LIN {X 0,Y 253.688,Z 332.355,A -85,B 0,C 180,E1 -18838.131,E2 -18838.131} C_VEL
LIN {X 0,Y 253.519,Z 331.287,A -85,B 0,C 180,E1 -18838.229,E2 -18838.229} C_VEL
LIN {X 0,Y 251.232,Z 319.885,A -85,B 0,C 180,E1 -18842.107,E2 -18842.107} C_VEL
LIN {X 0,Y 249.083,Z 309.456,A -85,B 0,C 180,E1 -18845.847,E2 -18845.847} C_VEL
LIN {X 0,Y 248.969,Z 309.472,A -85,B 0,C 180,E1 -18850.484,E2 -18850.484} C_VEL
LIN {X 0,Y 248.957,Z 309.474,A -85,B 0,C 180,E1 -18854.887,E2 -18854.887} C_VEL
LIN {X 0,Y 248.971,Z 309.47,A -85,B 0,C 180,E1 -18857.352,E2 -18857.352} C_VEL
LIN {X 0,Y 249.037,Z 309.461,A -85,B 0,C 180,E1 -18862.199,E2 -18862.199} C_VEL
LIN {X 0,Y 249.034,Z 309.462,A -85,B 0,C 180,E1 -18865.637,E2 -18865.637} C_VEL
LIN {X 0,Y 248.989,Z 309.469,A -85,B 0,C 180,E1 -18869.464,E2 -18869.464} C_VEL
LIN {X 0,Y 249.025,Z 309.467,A -85,B 0,C 180,E1 -18873.156,E2 -18873.156} C_VEL
LIN {X 0,Y 249.039,Z 309.461,A -85,B 0,C 180,E1 -18876.728,E2 -18876.728} C_VEL
LIN {X 0,Y 249.043,Z 309.46,A -85,B 0,C 180,E1 -18880.205,E2 -18880.205} C_VEL
LIN {X 0,Y 249.146,Z 309.448,A -85,B 0,C 180,E1 -18883.615,E2 -18883.615} C_VEL
LIN {X 0,Y 249.209,Z 309.44,A -85,B 0,C 180,E1 -18888.614,E2 -18888.614} C_VEL
LIN {X 0,Y 249.431,Z 309.412,A -85,B 0,C 180,E1 -18891.9,E2 -18891.9} C_VEL
LIN {X 0,Y 249.266,Z 309.434,A -85,B 0,C 180,E1 -18895.147,E2 -18895.147} C_VEL
LIN {X 0,Y 249.653,Z 309.385,A -85,B 0,C 180,E1 -18898.386,E2 -18898.386} C_VEL
LIN {X 0,Y 249.653,Z 309.386,A -85,B 0,C 180,E1 -18901.612,E2 -18901.612} C_VEL
LIN {X 0,Y 249.41,Z 309.413,A -85,B 0,C 180,E1 -18906.803,E2 -18906.803} C_VEL
LIN {X 0,Y 249.32,Z 309.427,A -85,B 0,C 180,E1 -18909.737,E2 -18909.737} C_VEL
LIN {X 0,Y 249.153,Z 309.447,A -85,B 0,C 180,E1 -18914.706,E2 -18914.706} C_VEL
LIN {X 0,Y 249.067,Z 309.457,A -85,B 0,C 180,E1 -18918.082,E2 -18918.082} C_VEL
LIN {X 0,Y 249.032,Z 309.464,A -85,B 0,C 180,E1 -18921.522,E2 -18921.522} C_VEL
LIN {X 0,Y 249.103,Z 309.455,A -85,B 0,C 180,E1 -18925.475,E2 -18925.475} C_VEL
LIN {X 0,Y 249.061,Z 309.457,A -85,B 0,C 180,E1 -18928.989,E2 -18928.989} C_VEL
LIN {X 0,Y 249.019,Z 309.464,A -85,B 0,C 180,E1 -18932.426,E2 -18932.426} C_VEL
LIN {X 0,Y 249.043,Z 309.461,A -85,B 0,C 180,E1 -18936.342,E2 -18936.342} C_VEL
LIN {X 0,Y 248.997,Z 309.467,A -85,B 0,C 180,E1 -18940.479,E2 -18940.479} C_VEL
LIN {X 0,Y 249.004,Z 309.464,A -85,B 0,C 180,E1 -18944.878,E2 -18944.878} C_VEL
LIN {X 0,Y 249.05,Z 309.46,A -85,B 0,C 180,E1 -18947.372,E2 -18947.372} C_VEL
LIN {X 0,Y 249.046,Z 309.46,A -85,B 0,C 180,E1 -18951.624,E2 -18951.624} C_VEL
LIN {X 0,Y 249.057,Z 309.459,A -85,B 0,C 180,E1 -18955.642,E2 -18955.642} C_VEL
LIN {X 0,Y 249.043,Z 309.46,A -85,B 0,C 180,E1 -18959.472,E2 -18959.472} C_VEL
LIN {X 0,Y 249.068,Z 309.457,A -85,B 0,C 180,E1 -18963.162,E2 -18963.162} C_VEL
LIN {X 0,Y 249.078,Z 309.457,A -85,B 0,C 180,E1 -18966.732,E2 -18966.732} C_VEL
LIN {X 0,Y 249.11,Z 309.453,A -85,B 0,C 180,E1 -18970.211,E2 -18970.211} C_VEL
LIN {X 0,Y 249.24,Z 309.436,A -85,B 0,C 180,E1 -18973.621,E2 -18973.621} C_VEL
LIN {X 0,Y 249.251,Z 309.437,A -85,B 0,C 180,E1 -18978.615,E2 -18978.615} C_VEL
LIN {X 0,Y 249.483,Z 309.406,A -85,B 0,C 180,E1 -18981.901,E2 -18981.901} C_VEL
LIN {X 0,Y 249.434,Z 309.414,A -85,B 0,C 180,E1 -18986.767,E2 -18986.767} C_VEL
LIN {X 0,Y 249.726,Z 309.376,A -85,B 0,C 180,E1 -18989.997,E2 -18989.997} C_VEL
LIN {X 0,Y 249.434,Z 309.411,A -85,B 0,C 180,E1 -18993.228,E2 -18993.228} C_VEL
LIN {X 0,Y 249.479,Z 309.407,A -85,B 0,C 180,E1 -18998.094,E2 -18998.094} C_VEL
LIN {X 0,Y 249.248,Z 309.435,A -85,B 0,C 180,E1 -19001.38,E2 -19001.38} C_VEL
LIN {X 0,Y 249.234,Z 309.437,A -85,B 0,C 180,E1 -19006.374,E2 -19006.374} C_VEL
LIN {X 0,Y 249.125,Z 309.451,A -85,B 0,C 180,E1 -19011.51,E2 -19011.51} C_VEL
LIN {X 0,Y 249.119,Z 309.452,A -85,B 0,C 180,E1 -19015.478,E2 -19015.478} C_VEL
LIN {X 0,Y 249.069,Z 309.461,A -85,B 0,C 180,E1 -19018.989,E2 -19018.989} C_VEL
LIN {X 0,Y 249.08,Z 309.458,A -85,B 0,C 180,E1 -19023.799,E2 -19023.799} C_VEL
LIN {X 0,Y 252.845,Z 319.658,A -85,B 0,C 180,E1 -19024.515,E2 -19024.515} C_VEL
LIN {X 0,Y 259.68,Z 338.346,A -85,B 0,C 180,E1 -19025.737,E2 -19025.737} C_VEL
LIN {X 0,Y 260.257,Z 340.087,A -85,B 0,C 180,E1 -19025.842,E2 -19025.842} C_VEL
LIN {X 0,Y 257.273,Z 412.228,A -85,B 0,C 180,E1 -19028.37,E2 -19028.37} C_VEL
LIN {X 0,Y 256.65,Z 424.844,A -85,B 0,C 180,E1 -19029.098,E2 -19029.098} C_VEL
LIN {X 0,Y 255.648,Z 437.472,A -85,B 0,C 180,E1 -19030.113,E2 -19030.113} C_VEL
LIN {X 0,Y 254.445,Z 449.649,A -85,B 0,C 180,E1 -19031.423,E2 -19031.423} C_VEL
LIN {X 0,Y 253.15,Z 460.66,A -85,B 0,C 180,E1 -19032.928,E2 -19032.928} C_VEL
LIN {X 0,Y 251.959,Z 470.882,A -85,B 0,C 180,E1 -19034.662,E2 -19034.662} C_VEL
LIN {X 0,Y 250.599,Z 481.033,A -85,B 0,C 180,E1 -19036.807,E2 -19036.807} C_VEL
LIN {X 0,Y 249.471,Z 489.721,A -85,B 0,C 180,E1 -19039.082,E2 -19039.082} C_VEL
LIN {X 0,Y 248.537,Z 497.225,A -85,B 0,C 180,E1 -19041.531,E2 -19041.531} C_VEL
LIN {X 0,Y 247.852,Z 503.12,A -85,B 0,C 180,E1 -19043.96,E2 -19043.96} C_VEL
LIN {X 0,Y 247.453,Z 507.724,A -85,B 0,C 180,E1 -19046.371,E2 -19046.371} C_VEL
LIN {X 0,Y 247.04,Z 511.734,A -85,B 0,C 180,E1 -19049.199,E2 -19049.199} C_VEL
LIN {X 0,Y 246.904,Z 514.316,A -85,B 0,C 180,E1 -19051.917,E2 -19051.917} C_VEL
LIN {X 0,Y 247.262,Z 515.891,A -85,B 0,C 180,E1 -19055.423,E2 -19055.423} C_VEL
LIN {X 0,Y 247.98,Z 515.755,A -85,B 0,C 180,E1 -19058.382,E2 -19058.382} C_VEL
LIN {X 0,Y 248.621,Z 515,A -85,B 0,C 180,E1 -19060.172,E2 -19060.172} C_VEL
LIN {X 0,Y 249.915,Z 512.823,A -85,B 0,C 180,E1 -19062.939,E2 -19062.939} C_VEL
LIN {X 0,Y 251.501,Z 509.738,A -85,B 0,C 180,E1 -19065.435,E2 -19065.435} C_VEL
LIN {X 0,Y 253.476,Z 505.327,A -85,B 0,C 180,E1 -19067.999,E2 -19067.999} C_VEL
LIN {X 0,Y 255.951,Z 499.537,A -85,B 0,C 180,E1 -19070.518,E2 -19070.518} C_VEL
LIN {X 0,Y 258.79,Z 492.2,A -85,B 0,C 180,E1 -19072.981,E2 -19072.981} C_VEL
LIN {X 0,Y 261.491,Z 484.692,A -85,B 0,C 180,E1 -19074.979,E2 -19074.979} C_VEL
LIN {X 0,Y 264.556,Z 475.406,A -85,B 0,C 180,E1 -19076.955,E2 -19076.955} C_VEL
LIN {X 0,Y 267.336,Z 465.509,A -85,B 0,C 180,E1 -19078.655,E2 -19078.655} C_VEL
LIN {X 0,Y 270.129,Z 454.102,A -85,B 0,C 180,E1 -19080.187,E2 -19080.187} C_VEL
LIN {X 0,Y 272.685,Z 441.841,A -85,B 0,C 180,E1 -19081.478,E2 -19081.478} C_VEL
LIN {X 0,Y 274.666,Z 429.131,A -85,B 0,C 180,E1 -19082.484,E2 -19082.484} C_VEL
LIN {X 0,Y 276.268,Z 415.345,A -85,B 0,C 180,E1 -19083.248,E2 -19083.248} C_VEL
LIN {X 0,Y 281,Z 357.266,A -85,B 0,C 180,E1 -19085.293,E2 -19085.293} C_VEL
LIN {X 0,Y 277.332,Z 349.628,A -85,B 0,C 180,E1 -19086.613,E2 -19086.613} C_VEL
LIN {X 0,Y 276.385,Z 347.949,A -85,B 0,C 180,E1 -19086.951,E2 -19086.951} C_VEL
LIN {X 0,Y 274.604,Z 345.866,A -85,B 0,C 180,E1 -19087.543,E2 -19087.543} C_VEL
LIN {X 0,Y 270.87,Z 344.364,A -85,B 0,C 180,E1 -19088.684,E2 -19088.684} C_VEL
LIN {X 0,Y 267.23,Z 343.003,A -85,B 0,C 180,E1 -19089.882,E2 -19089.882} C_VEL
LIN {X 0,Y 265.578,Z 341.11,A -85,B 0,C 180,E1 -19090.553,E2 -19090.553} C_VEL
LIN {X 0,Y 262.045,Z 336.05,A -85,B 0,C 180,E1 -19092.207,E2 -19092.207} C_VEL
LIN {X 0,Y 258.278,Z 331.025,A -85,B 0,C 180,E1 -19094.177,E2 -19094.177} C_VEL
LIN {X 0,Y 254.479,Z 326.181,A -85,B 0,C 180,E1 -19096.472,E2 -19096.472} C_VEL
LIN {X 0,Y 251.933,Z 323.447,A -85,B 0,C 180,E1 -19098.228,E2 -19098.228} C_VEL
LIN {X 0,Y 248.642,Z 319.476,A -85,B 0,C 180,E1 -19101.152,E2 -19101.152} C_VEL
LIN {X 0,Y 244.923,Z 316.459,A -85,B 0,C 180,E1 -19106.218,E2 -19106.218} C_VEL
LIN {X 0,Y 244.041,Z 315.707,A -85,B 0,C 180,E1 -19109.432,E2 -19109.432} C_VEL
LIN {X 0,Y 244.605,Z 316.843,A -85,B 0,C 180,E1 -19113.582,E2 -19113.582} C_VEL
LIN {X 0,Y 245.437,Z 318.272,A -85,B 0,C 180,E1 -19116.185,E2 -19116.185} C_VEL
LIN {X 0,Y 248.579,Z 323.493,A -85,B 0,C 180,E1 -19120.431,E2 -19120.431} C_VEL
LIN {X 0,Y 251.56,Z 327.54,A -85,B 0,C 180,E1 -19123.051,E2 -19123.051} C_VEL
LIN {X 0,Y 256.502,Z 335.172,A -85,B 0,C 180,E1 -19126.428,E2 -19126.428} C_VEL
LIN {X 0,Y 260.53,Z 342.026,A -85,B 0,C 180,E1 -19128.71,E2 -19128.71} C_VEL
LIN {X 0,Y 263.954,Z 348.304,A -85,B 0,C 180,E1 -19130.433,E2 -19130.433} C_VEL
LIN {X 0,Y 267.188,Z 354.826,A -85,B 0,C 180,E1 -19131.92,E2 -19131.92} C_VEL
LIN {X 0,Y 270.159,Z 361.496,A -85,B 0,C 180,E1 -19133.236,E2 -19133.236} C_VEL
LIN {X 0,Y 272.398,Z 367.573,A -85,B 0,C 180,E1 -19134.204,E2 -19134.204} C_VEL
LIN {X 0,Y 273.727,Z 381.745,A -85,B 0,C 180,E1 -19135.364,E2 -19135.364} C_VEL
LIN {X 0,Y 274.04,Z 390.294,A -85,B 0,C 180,E1 -19135.927,E2 -19135.927} C_VEL
LIN {X 0,Y 269.906,Z 437.588,A -85,B 0,C 180,E1 -19137.634,E2 -19137.634} C_VEL
LIN {X 0,Y 267.932,Z 451.025,A -85,B 0,C 180,E1 -19138.364,E2 -19138.364} C_VEL
LIN {X 0,Y 265.251,Z 463.95,A -85,B 0,C 180,E1 -19139.34,E2 -19139.34} C_VEL
LIN {X 0,Y 262.356,Z 475.61,A -85,B 0,C 180,E1 -19140.519,E2 -19140.519} C_VEL
LIN {X 0,Y 259.28,Z 486.361,A -85,B 0,C 180,E1 -19141.909,E2 -19141.909} C_VEL
LIN {X 0,Y 255.526,Z 498.244,A -85,B 0,C 180,E1 -19143.898,E2 -19143.898} C_VEL
LIN {X 0,Y 252.405,Z 507.111,A -85,B 0,C 180,E1 -19145.757,E2 -19145.757} C_VEL
LIN {X 0,Y 249.187,Z 515.851,A -85,B 0,C 180,E1 -19148.061,E2 -19148.061} C_VEL
LIN {X 0,Y 246.082,Z 523.981,A -85,B 0,C 180,E1 -19150.831,E2 -19150.831} C_VEL
LIN {X 0,Y 244.064,Z 529.572,A -85,B 0,C 180,E1 -19153.269,E2 -19153.269} C_VEL
LIN {X 0,Y 242.205,Z 534.014,A -85,B 0,C 180,E1 -19155.725,E2 -19155.725} C_VEL
LIN {X 0,Y 241.026,Z 537.398,A -85,B 0,C 180,E1 -19158.226,E2 -19158.226} C_VEL
LIN {X 0,Y 240.501,Z 539.133,A -85,B 0,C 180,E1 -19159.906,E2 -19159.906} C_VEL
LIN {X 0,Y 240.145,Z 540.433,A -85,B 0,C 180,E1 -19161.589,E2 -19161.589} C_VEL
LIN {X 0,Y 239.914,Z 541.794,A -85,B 0,C 180,E1 -19164.876,E2 -19164.876} C_VEL
LIN {X 0,Y 240.011,Z 541.905,A -85,B 0,C 180,E1 -19166.646,E2 -19166.646} C_VEL
LIN {X 0,Y 240.056,Z 541.562,A -85,B 0,C 180,E1 -19168.325,E2 -19168.325} C_VEL
LIN {X 0,Y 240.251,Z 540.779,A -85,B 0,C 180,E1 -19170.003,E2 -19170.003} C_VEL
LIN {X 0,Y 240.131,Z 539.542,A -85,B 0,C 180,E1 -19171.68,E2 -19171.68} C_VEL
LIN {X 0,Y 240.193,Z 536.83,A -85,B 0,C 180,E1 -19174.197,E2 -19174.197} C_VEL
LIN {X 0,Y 240.192,Z 532.978,A -85,B 0,C 180,E1 -19176.723,E2 -19176.723} C_VEL
LIN {X 0,Y 240.41,Z 527.9,A -85,B 0,C 180,E1 -19179.254,E2 -19179.254} C_VEL
LIN {X 0,Y 240.928,Z 521.439,A -85,B 0,C 180,E1 -19181.784,E2 -19181.784} C_VEL
LIN {X 0,Y 241.908,Z 513.277,A -85,B 0,C 180,E1 -19184.298,E2 -19184.298} C_VEL
LIN {X 0,Y 242.966,Z 504.922,A -85,B 0,C 180,E1 -19186.382,E2 -19186.382} C_VEL
LIN {X 0,Y 244.331,Z 494.733,A -85,B 0,C 180,E1 -19188.447,E2 -19188.447} C_VEL
LIN {X 0,Y 245.863,Z 483.261,A -85,B 0,C 180,E1 -19190.28,E2 -19190.28} C_VEL
LIN {X 0,Y 247.151,Z 472.105,A -85,B 0,C 180,E1 -19191.696,E2 -19191.696} C_VEL
LIN {X 0,Y 248.519,Z 459.905,A -85,B 0,C 180,E1 -19192.883,E2 -19192.883} C_VEL
LIN {X 0,Y 249.739,Z 445.91,A -85,B 0,C 180,E1 -19193.862,E2 -19193.862} C_VEL
LIN {X 0,Y 250.331,Z 432.886,A -85,B 0,C 180,E1 -19194.463,E2 -19194.463} C_VEL
LIN {X 0,Y 252.364,Z 383.36,A -85,B 0,C 180,E1 -19196.236,E2 -19196.236} C_VEL
LIN {X 0,Y 247.119,Z 334.2,A -85,B 0,C 180,E1 -19198.56,E2 -19198.56} C_VEL
LIN {X 0,Y 246.261,Z 331.04,A -85,B 0,C 180,E1 -19198.763,E2 -19198.763} C_VEL
LIN {X 0,Y 243.683,Z 318.326,A -85,B 0,C 180,E1 -19203.239,E2 -19203.239} C_VEL
LIN {X 0,Y 242.055,Z 310.332,A -85,B 0,C 180,E1 -19206.209,E2 -19206.209} C_VEL
LIN {X 0,Y 241.896,Z 310.355,A -85,B 0,C 180,E1 -19210.939,E2 -19210.939} C_VEL
LIN {X 0,Y 241.891,Z 310.352,A -85,B 0,C 180,E1 -19214.209,E2 -19214.209} C_VEL
LIN {X 0,Y 241.901,Z 310.35,A -85,B 0,C 180,E1 -19218.069,E2 -19218.069} C_VEL
LIN {X 0,Y 241.977,Z 310.341,A -85,B 0,C 180,E1 -19222.415,E2 -19222.415} C_VEL
LIN {X 0,Y 241.96,Z 310.344,A -85,B 0,C 180,E1 -19226.503,E2 -19226.503} C_VEL
LIN {X 0,Y 241.968,Z 310.343,A -85,B 0,C 180,E1 -19230.612,E2 -19230.612} C_VEL
LIN {X 0,Y 242.024,Z 310.335,A -85,B 0,C 180,E1 -19234.177,E2 -19234.177} C_VEL
LIN {X 0,Y 241.98,Z 310.339,A -85,B 0,C 180,E1 -19238.334,E2 -19238.334} C_VEL
LIN {X 0,Y 242.103,Z 310.328,A -85,B 0,C 180,E1 -19243.317,E2 -19243.317} C_VEL
LIN {X 0,Y 242.145,Z 310.32,A -85,B 0,C 180,E1 -19248.277,E2 -19248.277} C_VEL
LIN {X 0,Y 242.378,Z 310.292,A -85,B 0,C 180,E1 -19251.663,E2 -19251.663} C_VEL
LIN {X 0,Y 242.401,Z 310.29,A -85,B 0,C 180,E1 -19253.339,E2 -19253.339} C_VEL
LIN {X 0,Y 242.614,Z 310.262,A -85,B 0,C 180,E1 -19258.339,E2 -19258.339} C_VEL
LIN {X 0,Y 242.614,Z 310.262,A -85,B 0,C 180,E1 -19261.659,E2 -19261.659} C_VEL
LIN {X 0,Y 242.389,Z 310.289,A -85,B 0,C 180,E1 -19266.778,E2 -19266.778} C_VEL
LIN {X 0,Y 242.248,Z 310.306,A -85,B 0,C 180,E1 -19270.024,E2 -19270.024} C_VEL
LIN {X 0,Y 242.105,Z 310.326,A -85,B 0,C 180,E1 -19275.144,E2 -19275.144} C_VEL
LIN {X 0,Y 242.005,Z 310.335,A -85,B 0,C 180,E1 -19278.629,E2 -19278.629} C_VEL
LIN {X 0,Y 241.975,Z 310.343,A -85,B 0,C 180,E1 -19282.183,E2 -19282.183} C_VEL
LIN {X 0,Y 242.056,Z 310.333,A -85,B 0,C 180,E1 -19285.838,E2 -19285.838} C_VEL
LIN {X 0,Y 241.996,Z 310.34,A -85,B 0,C 180,E1 -19289.584,E2 -19289.584} C_VEL
LIN {X 0,Y 241.971,Z 310.343,A -85,B 0,C 180,E1 -19293.493,E2 -19293.493} C_VEL
LIN {X 0,Y 241.983,Z 310.34,A -85,B 0,C 180,E1 -19297.582,E2 -19297.582} C_VEL
LIN {X 0,Y 241.931,Z 310.35,A -85,B 0,C 180,E1 -19301.923,E2 -19301.923} C_VEL
LIN {X 0,Y 241.979,Z 310.342,A -85,B 0,C 180,E1 -19306.559,E2 -19306.559} C_VEL
LIN {X 0,Y 242.002,Z 310.34,A -85,B 0,C 180,E1 -19310.291,E2 -19310.291} C_VEL
LIN {X 0,Y 242.033,Z 310.336,A -85,B 0,C 180,E1 -19314.498,E2 -19314.498} C_VEL
LIN {X 0,Y 241.97,Z 310.344,A -85,B 0,C 180,E1 -19318.48,E2 -19318.48} C_VEL
LIN {X 0,Y 241.999,Z 310.34,A -85,B 0,C 180,E1 -19322.312,E2 -19322.312} C_VEL
LIN {X 0,Y 242.056,Z 310.333,A -85,B 0,C 180,E1 -19326.015,E2 -19326.015} C_VEL
LIN {X 0,Y 242.036,Z 310.331,A -85,B 0,C 180,E1 -19329.607,E2 -19329.607} C_VEL
LIN {X 0,Y 242.162,Z 310.318,A -85,B 0,C 180,E1 -19333.277,E2 -19333.277} C_VEL
LIN {X 0,Y 242.185,Z 310.316,A -85,B 0,C 180,E1 -19338.278,E2 -19338.278} C_VEL
LIN {X 0,Y 242.433,Z 310.284,A -85,B 0,C 180,E1 -19341.664,E2 -19341.664} C_VEL
LIN {X 0,Y 242.258,Z 310.305,A -85,B 0,C 180,E1 -19345.005,E2 -19345.005} C_VEL
LIN {X 0,Y 242.634,Z 310.26,A -85,B 0,C 180,E1 -19348.338,E2 -19348.338} C_VEL
LIN {X 0,Y 242.634,Z 310.259,A -85,B 0,C 180,E1 -19351.657,E2 -19351.657} C_VEL
LIN {X 0,Y 242.429,Z 310.288,A -85,B 0,C 180,E1 -19356.656,E2 -19356.656} C_VEL
LIN {X 0,Y 242.34,Z 310.296,A -85,B 0,C 180,E1 -19360.017,E2 -19360.017} C_VEL
LIN {X 0,Y 242.16,Z 310.319,A -85,B 0,C 180,E1 -19365.137,E2 -19365.137} C_VEL
LIN {X 0,Y 242.081,Z 310.33,A -85,B 0,C 180,E1 -19368.619,E2 -19368.619} C_VEL
LIN {X 0,Y 242.053,Z 310.331,A -85,B 0,C 180,E1 -19372.171,E2 -19372.171} C_VEL
LIN {X 0,Y 242.054,Z 310.331,A -85,B 0,C 180,E1 -19375.834,E2 -19375.834} C_VEL
LIN {X 0,Y 242.016,Z 310.338,A -85,B 0,C 180,E1 -19379.576,E2 -19379.576} C_VEL
LIN {X 0,Y 241.996,Z 310.344,A -85,B 0,C 180,E1 -19383.273,E2 -19383.273} C_VEL
LIN {X 0,Y 252.994,Z 339.978,A -85,B 0,C 180,E1 -19385.314,E2 -19385.314} C_VEL
LIN {X 0,Y 253.374,Z 342.402,A -85,B 0,C 180,E1 -19385.436,E2 -19385.436} C_VEL
LIN {X 0,Y 250.392,Z 412.965,A -85,B 0,C 180,E1 -19387.993,E2 -19387.993} C_VEL
LIN {X 0,Y 249.686,Z 426.336,A -85,B 0,C 180,E1 -19388.802,E2 -19388.802} C_VEL
LIN {X 0,Y 248.688,Z 438.197,A -85,B 0,C 180,E1 -19389.797,E2 -19389.797} C_VEL
LIN {X 0,Y 247.454,Z 450.568,A -85,B 0,C 180,E1 -19391.182,E2 -19391.182} C_VEL
LIN {X 0,Y 246.031,Z 462.066,A -85,B 0,C 180,E1 -19392.821,E2 -19392.821} C_VEL
LIN {X 0,Y 244.739,Z 472.544,A -85,B 0,C 180,E1 -19394.701,E2 -19394.701} C_VEL
LIN {X 0,Y 243.387,Z 482.763,A -85,B 0,C 180,E1 -19396.986,E2 -19396.986} C_VEL
LIN {X 0,Y 242.272,Z 490.914,A -85,B 0,C 180,E1 -19399.239,E2 -19399.239} C_VEL
LIN {X 0,Y 241.333,Z 498.388,A -85,B 0,C 180,E1 -19401.828,E2 -19401.828} C_VEL
LIN {X 0,Y 240.681,Z 504.014,A -85,B 0,C 180,E1 -19404.268,E2 -19404.268} C_VEL
LIN {X 0,Y 240.219,Z 509.293,A -85,B 0,C 180,E1 -19407.233,E2 -19407.233} C_VEL
LIN {X 0,Y 239.86,Z 512.936,A -85,B 0,C 180,E1 -19410.126,E2 -19410.126} C_VEL
LIN {X 0,Y 239.809,Z 514.611,A -85,B 0,C 180,E1 -19412.038,E2 -19412.038} C_VEL
LIN {X 0,Y 240.131,Z 516.193,A -85,B 0,C 180,E1 -19415.114,E2 -19415.114} C_VEL
LIN {X 0,Y 240.672,Z 516.431,A -85,B 0,C 180,E1 -19417.691,E2 -19417.691} C_VEL
LIN {X 0,Y 241.307,Z 515.986,A -85,B 0,C 180,E1 -19419.544,E2 -19419.544} C_VEL
LIN {X 0,Y 242.747,Z 514.007,A -85,B 0,C 180,E1 -19422.799,E2 -19422.799} C_VEL
LIN {X 0,Y 244.697,Z 510.583,A -85,B 0,C 180,E1 -19425.87,E2 -19425.87} C_VEL
LIN {X 0,Y 246.788,Z 506.294,A -85,B 0,C 180,E1 -19428.502,E2 -19428.502} C_VEL
LIN {X 0,Y 249.129,Z 501.304,A -85,B 0,C 180,E1 -19430.827,E2 -19430.827} C_VEL
LIN {X 0,Y 251.883,Z 494.84,A -85,B 0,C 180,E1 -19433.19,E2 -19433.19} C_VEL
LIN {X 0,Y 255.266,Z 486.167,A -85,B 0,C 180,E1 -19435.659,E2 -19435.659} C_VEL
LIN {X 0,Y 258.464,Z 477.097,A -85,B 0,C 180,E1 -19437.663,E2 -19437.663} C_VEL
LIN {X 0,Y 261.397,Z 467.526,A -85,B 0,C 180,E1 -19439.395,E2 -19439.395} C_VEL
LIN {X 0,Y 264.333,Z 456.654,A -85,B 0,C 180,E1 -19440.953,E2 -19440.953} C_VEL
LIN {X 0,Y 267.118,Z 444.188,A -85,B 0,C 180,E1 -19442.331,E2 -19442.331} C_VEL
LIN {X 0,Y 269.308,Z 431.823,A -85,B 0,C 180,E1 -19443.367,E2 -19443.367} C_VEL
LIN {X 0,Y 270.946,Z 419.021,A -85,B 0,C 180,E1 -19444.138,E2 -19444.138} C_VEL
LIN {X 0,Y 273.353,Z 391.394,A -85,B 0,C 180,E1 -19445.196,E2 -19445.196} C_VEL
LIN {X 0,Y 276.123,Z 360.168,A -85,B 0,C 180,E1 -19446.306,E2 -19446.306} C_VEL
LIN {X 0,Y 273.4,Z 354.391,A -85,B 0,C 180,E1 -19447.344,E2 -19447.344} C_VEL
LIN {X 0,Y 266.645,Z 342.828,A -85,B 0,C 180,E1 -19450.078,E2 -19450.078} C_VEL
LIN {X 0,Y 265.578,Z 341.11,A -85,B 0,C 180,E1 -19450.553,E2 -19450.553} C_VEL
LIN {X 0,Y 264.177,Z 339.037,A -85,B 0,C 180,E1 -19451.2,E2 -19451.2} C_VEL
LIN {X 0,Y 261.646,Z 337.151,A -85,B 0,C 180,E1 -19452.286,E2 -19452.286} C_VEL
LIN {X 0,Y 255.468,Z 335.207,A -85,B 0,C 180,E1 -19455.07,E2 -19455.07} C_VEL
LIN {X 0,Y 253.285,Z 333.784,A -85,B 0,C 180,E1 -19456.303,E2 -19456.303} C_VEL
LIN {X 0,Y 252.689,Z 333.04,A -85,B 0,C 180,E1 -19456.706,E2 -19456.706} C_VEL
LIN {X 0,Y 250.034,Z 330.073,A -85,B 0,C 180,E1 -19458.609,E2 -19458.609} C_VEL
LIN {X 0,Y 247.051,Z 326.377,A -85,B 0,C 180,E1 -19461.369,E2 -19461.369} C_VEL
LIN {X 0,Y 243.656,Z 323.483,A -85,B 0,C 180,E1 -19466.141,E2 -19466.141} C_VEL
LIN {X 0,Y 242.898,Z 322.75,A -85,B 0,C 180,E1 -19468.441,E2 -19468.441} C_VEL
LIN {X 0,Y 242.635,Z 323.055,A -85,B 0,C 180,E1 -19471.425,E2 -19471.425} C_VEL
LIN {X 0,Y 243.828,Z 324.749,A -85,B 0,C 180,E1 -19475.597,E2 -19475.597} C_VEL
LIN {X 0,Y 246.834,Z 330.215,A -85,B 0,C 180,E1 -19480.073,E2 -19480.073} C_VEL
LIN {X 0,Y 249.476,Z 333.985,A -85,B 0,C 180,E1 -19482.541,E2 -19482.541} C_VEL
LIN {X 0,Y 254.034,Z 341.357,A -85,B 0,C 180,E1 -19485.863,E2 -19485.863} C_VEL
LIN {X 0,Y 257.599,Z 347.719,A -85,B 0,C 180,E1 -19488.032,E2 -19488.032} C_VEL
LIN {X 0,Y 260.823,Z 353.84,A -85,B 0,C 180,E1 -19489.742,E2 -19489.742} C_VEL
LIN {X 0,Y 264.614,Z 361.832,A -85,B 0,C 180,E1 -19491.605,E2 -19491.605} C_VEL
LIN {X 0,Y 268.022,Z 370.725,A -85,B 0,C 180,E1 -19493.214,E2 -19493.214} C_VEL
LIN {X 0,Y 269.139,Z 384.639,A -85,B 0,C 180,E1 -19494.376,E2 -19494.376} C_VEL
LIN {X 0,Y 269.345,Z 391.221,A -85,B 0,C 180,E1 -19494.82,E2 -19494.82} C_VEL
LIN {X 0,Y 265.149,Z 436.293,A -85,B 0,C 180,E1 -19496.469,E2 -19496.469} C_VEL
LIN {X 0,Y 262.983,Z 450.412,A -85,B 0,C 180,E1 -19497.244,E2 -19497.244} C_VEL
LIN {X 0,Y 260.193,Z 463.305,A -85,B 0,C 180,E1 -19498.223,E2 -19498.223} C_VEL
LIN {X 0,Y 256.756,Z 476.515,A -85,B 0,C 180,E1 -19499.583,E2 -19499.583} C_VEL
LIN {X 0,Y 253.544,Z 486.982,A -85,B 0,C 180,E1 -19500.988,E2 -19500.988} C_VEL
LIN {X 0,Y 249.948,Z 497.646,A -85,B 0,C 180,E1 -19502.818,E2 -19502.818} C_VEL
LIN {X 0,Y 246.61,Z 506.468,A -85,B 0,C 180,E1 -19504.698,E2 -19504.698} C_VEL
LIN {X 0,Y 243.209,Z 515.228,A -85,B 0,C 180,E1 -19507.044,E2 -19507.044} C_VEL
LIN {X 0,Y 240.268,Z 522.35,A -85,B 0,C 180,E1 -19509.456,E2 -19509.456} C_VEL
LIN {X 0,Y 237.975,Z 528.131,A -85,B 0,C 180,E1 -19511.94,E2 -19511.94} C_VEL
LIN {X 0,Y 235.908,Z 532.758,A -85,B 0,C 180,E1 -19514.452,E2 -19514.452} C_VEL
LIN {X 0,Y 234.372,Z 536.349,A -85,B 0,C 180,E1 -19517.007,E2 -19517.007} C_VEL
LIN {X 0,Y 233.483,Z 538.969,A -85,B 0,C 180,E1 -19519.599,E2 -19519.599} C_VEL
LIN {X 0,Y 232.901,Z 540.997,A -85,B 0,C 180,E1 -19523.071,E2 -19523.071} C_VEL
LIN {X 0,Y 232.846,Z 541.442,A -85,B 0,C 180,E1 -19524.909,E2 -19524.909} C_VEL
LIN {X 0,Y 232.921,Z 541.435,A -85,B 0,C 180,E1 -19526.543,E2 -19526.543} C_VEL
LIN {X 0,Y 232.982,Z 540.997,A -85,B 0,C 180,E1 -19528.274,E2 -19528.274} C_VEL
LIN {X 0,Y 233.172,Z 540.152,A -85,B 0,C 180,E1 -19530.003,E2 -19530.003} C_VEL
LIN {X 0,Y 233.057,Z 538.853,A -85,B 0,C 180,E1 -19531.731,E2 -19531.731} C_VEL
LIN {X 0,Y 233.138,Z 536.01,A -85,B 0,C 180,E1 -19534.324,E2 -19534.324} C_VEL
LIN {X 0,Y 233.133,Z 532.013,A -85,B 0,C 180,E1 -19536.928,E2 -19536.928} C_VEL
LIN {X 0,Y 233.433,Z 525.73,A -85,B 0,C 180,E1 -19539.971,E2 -19539.971} C_VEL
LIN {X 0,Y 234.082,Z 518.804,A -85,B 0,C 180,E1 -19542.574,E2 -19542.574} C_VEL
LIN {X 0,Y 235.175,Z 510.139,A -85,B 0,C 180,E1 -19545.16,E2 -19545.16} C_VEL
LIN {X 0,Y 236.305,Z 501.171,A -85,B 0,C 180,E1 -19547.303,E2 -19547.303} C_VEL
LIN {X 0,Y 237.879,Z 490.215,A -85,B 0,C 180,E1 -19549.414,E2 -19549.414} C_VEL
LIN {X 0,Y 239.303,Z 479.213,A -85,B 0,C 180,E1 -19551.086,E2 -19551.086} C_VEL
LIN {X 0,Y 240.749,Z 467.112,A -85,B 0,C 180,E1 -19552.529,E2 -19552.529} C_VEL
LIN {X 0,Y 242.073,Z 454.752,A -85,B 0,C 180,E1 -19553.642,E2 -19553.642} C_VEL
LIN {X 0,Y 243.227,Z 440.281,A -85,B 0,C 180,E1 -19554.542,E2 -19554.542} C_VEL
LIN {X 0,Y 245.458,Z 383.245,A -85,B 0,C 180,E1 -19556.715,E2 -19556.715} C_VEL
LIN {X 0,Y 240.428,Z 335.664,A -85,B 0,C 180,E1 -19559.029,E2 -19559.029} C_VEL
LIN {X 0,Y 238.941,Z 330.57,A -85,B 0,C 180,E1 -19559.393,E2 -19559.393} C_VEL
LIN {X 0,Y 236.543,Z 318.716,A -85,B 0,C 180,E1 -19563.703,E2 -19563.703} C_VEL
LIN {X 0,Y 235,Z 311.211,A -85,B 0,C 180,E1 -19566.555,E2 -19566.555} C_VEL
LIN {X 0,Y 234.846,Z 311.231,A -85,B 0,C 180,E1 -19571.174,E2 -19571.174} C_VEL
LIN {X 0,Y 234.857,Z 311.225,A -85,B 0,C 180,E1 -19575.903,E2 -19575.903} C_VEL
LIN {X 0,Y 234.848,Z 311.232,A -85,B 0,C 180,E1 -19578.824,E2 -19578.824} C_VEL
LIN {X 0,Y 234.914,Z 311.224,A -85,B 0,C 180,E1 -19581.077,E2 -19581.077} C_VEL
LIN {X 0,Y 234.892,Z 311.225,A -85,B 0,C 180,E1 -19585.355,E2 -19585.355} C_VEL
LIN {X 0,Y 234.882,Z 311.226,A -85,B 0,C 180,E1 -19589.424,E2 -19589.424} C_VEL
LIN {X 0,Y 234.961,Z 311.215,A -85,B 0,C 180,E1 -19593.805,E2 -19593.805} C_VEL
LIN {X 0,Y 234.954,Z 311.214,A -85,B 0,C 180,E1 -19598.007,E2 -19598.007} C_VEL
LIN {X 0,Y 235.044,Z 311.208,A -85,B 0,C 180,E1 -19603.092,E2 -19603.092} C_VEL
LIN {X 0,Y 235.079,Z 311.201,A -85,B 0,C 180,E1 -19607.919,E2 -19607.919} C_VEL
LIN {X 0,Y 235.307,Z 311.175,A -85,B 0,C 180,E1 -19611.411,E2 -19611.411} C_VEL
LIN {X 0,Y 235.351,Z 311.168,A -85,B 0,C 180,E1 -19613.139,E2 -19613.139} C_VEL
LIN {X 0,Y 235.574,Z 311.139,A -85,B 0,C 180,E1 -19618.29,E2 -19618.29} C_VEL
LIN {X 0,Y 235.574,Z 311.139,A -85,B 0,C 180,E1 -19621.709,E2 -19621.709} C_VEL
LIN {X 0,Y 235.348,Z 311.167,A -85,B 0,C 180,E1 -19626.859,E2 -19626.859} C_VEL
LIN {X 0,Y 235.197,Z 311.183,A -85,B 0,C 180,E1 -19630.327,E2 -19630.327} C_VEL
LIN {X 0,Y 235.055,Z 311.207,A -85,B 0,C 180,E1 -19635.609,E2 -19635.609} C_VEL
LIN {X 0,Y 234.947,Z 311.215,A -85,B 0,C 180,E1 -19639.21,E2 -19639.21} C_VEL
LIN {X 0,Y 234.93,Z 311.219,A -85,B 0,C 180,E1 -19642.885,E2 -19642.885} C_VEL
LIN {X 0,Y 234.956,Z 311.213,A -85,B 0,C 180,E1 -19646.658,E2 -19646.658} C_VEL
LIN {X 0,Y 234.911,Z 311.221,A -85,B 0,C 180,E1 -19650.57,E2 -19650.57} C_VEL
LIN {X 0,Y 234.923,Z 311.218,A -85,B 0,C 180,E1 -19654.638,E2 -19654.638} C_VEL
LIN {X 0,Y 234.934,Z 311.218,A -85,B 0,C 180,E1 -19658.945,E2 -19658.945} C_VEL
LIN {X 0,Y 234.883,Z 311.224,A -85,B 0,C 180,E1 -19663.486,E2 -19663.486} C_VEL
LIN {X 0,Y 234.953,Z 311.217,A -85,B 0,C 180,E1 -19666.531,E2 -19666.531} C_VEL
LIN {X 0,Y 234.95,Z 311.215,A -85,B 0,C 180,E1 -19671.086,E2 -19671.086} C_VEL
LIN {X 0,Y 234.956,Z 311.215,A -85,B 0,C 180,E1 -19675.367,E2 -19675.367} C_VEL
LIN {X 0,Y 234.919,Z 311.219,A -85,B 0,C 180,E1 -19679.431,E2 -19679.431} C_VEL
LIN {X 0,Y 234.991,Z 311.212,A -85,B 0,C 180,E1 -19683.794,E2 -19683.794} C_VEL
LIN {X 0,Y 235.01,Z 311.207,A -85,B 0,C 180,E1 -19688.969,E2 -19688.969} C_VEL
LIN {X 0,Y 235.095,Z 311.199,A -85,B 0,C 180,E1 -19693.058,E2 -19693.058} C_VEL
LIN {X 0,Y 235.117,Z 311.194,A -85,B 0,C 180,E1 -19697.921,E2 -19697.921} C_VEL
LIN {X 0,Y 235.389,Z 311.162,A -85,B 0,C 180,E1 -19701.413,E2 -19701.413} C_VEL
LIN {X 0,Y 235.404,Z 311.16,A -85,B 0,C 180,E1 -19703.139,E2 -19703.139} C_VEL
LIN {X 0,Y 235.594,Z 311.137,A -85,B 0,C 180,E1 -19708.288,E2 -19708.288} C_VEL
LIN {X 0,Y 235.594,Z 311.136,A -85,B 0,C 180,E1 -19711.707,E2 -19711.707} C_VEL
LIN {X 0,Y 235.401,Z 311.164,A -85,B 0,C 180,E1 -19716.855,E2 -19716.855} C_VEL
LIN {X 0,Y 235.248,Z 311.18,A -85,B 0,C 180,E1 -19720.322,E2 -19720.322} C_VEL
LIN {X 0,Y 235.107,Z 311.195,A -85,B 0,C 180,E1 -19725.602,E2 -19725.602} C_VEL
LIN {X 0,Y 235.021,Z 311.211,A -85,B 0,C 180,E1 -19729.2,E2 -19729.2} C_VEL
LIN {X 0,Y 234.979,Z 311.215,A -85,B 0,C 180,E1 -19732.876,E2 -19732.876} C_VEL
LIN {X 0,Y 234.957,Z 311.217,A -85,B 0,C 180,E1 -19736.653,E2 -19736.653} C_VEL
LIN {X 0,Y 234.912,Z 311.223,A -85,B 0,C 180,E1 -19740.564,E2 -19740.564} C_VEL
LIN {X 0,Y 234.953,Z 311.277,A -85,B 0,C 180,E1 -19742.72,E2 -19742.72} C_VEL
LIN {X 0,Y 246.383,Z 341.938,A -85,B 0,C 180,E1 -19744.902,E2 -19744.902} C_VEL
LIN {X 0,Y 246.485,Z 346.089,A -85,B 0,C 180,E1 -19745.075,E2 -19745.075} C_VEL
LIN {X 0,Y 243.529,Z 412.847,A -85,B 0,C 180,E1 -19747.576,E2 -19747.576} C_VEL
LIN {X 0,Y 242.894,Z 425.09,A -85,B 0,C 180,E1 -19748.32,E2 -19748.32} C_VEL
LIN {X 0,Y 241.785,Z 438.101,A -85,B 0,C 180,E1 -19749.417,E2 -19749.417} C_VEL
LIN {X 0,Y 240.477,Z 450.806,A -85,B 0,C 180,E1 -19750.869,E2 -19750.869} C_VEL
LIN {X 0,Y 238.944,Z 463.039,A -85,B 0,C 180,E1 -19752.667,E2 -19752.667} C_VEL
LIN {X 0,Y 237.518,Z 474.118,A -85,B 0,C 180,E1 -19754.755,E2 -19754.755} C_VEL
LIN {X 0,Y 236.315,Z 483.106,A -85,B 0,C 180,E1 -19756.843,E2 -19756.843} C_VEL
LIN {X 0,Y 235.286,Z 490.477,A -85,B 0,C 180,E1 -19758.919,E2 -19758.919} C_VEL
LIN {X 0,Y 234.285,Z 498.385,A -85,B 0,C 180,E1 -19761.673,E2 -19761.673} C_VEL
LIN {X 0,Y 233.567,Z 504.368,A -85,B 0,C 180,E1 -19764.321,E2 -19764.321} C_VEL
LIN {X 0,Y 233.129,Z 509.3,A -85,B 0,C 180,E1 -19767.138,E2 -19767.138} C_VEL
LIN {X 0,Y 232.776,Z 513.104,A -85,B 0,C 180,E1 -19770.122,E2 -19770.122} C_VEL
LIN {X 0,Y 232.781,Z 515.522,A -85,B 0,C 180,E1 -19773.073,E2 -19773.073} C_VEL
LIN {X 0,Y 233.029,Z 516.444,A -85,B 0,C 180,E1 -19775.026,E2 -19775.026} C_VEL
LIN {X 0,Y 233.388,Z 516.887,A -85,B 0,C 180,E1 -19776.955,E2 -19776.955} C_VEL
LIN {X 0,Y 233.948,Z 516.768,A -85,B 0,C 180,E1 -19778.871,E2 -19778.871} C_VEL
LIN {X 0,Y 234.673,Z 516.183,A -85,B 0,C 180,E1 -19780.767,E2 -19780.767} C_VEL
LIN {X 0,Y 235.563,Z 515.086,A -85,B 0,C 180,E1 -19782.664,E2 -19782.664} C_VEL
LIN {X 0,Y 237.239,Z 512.539,A -85,B 0,C 180,E1 -19785.417,E2 -19785.417} C_VEL
LIN {X 0,Y 239.364,Z 508.813,A -85,B 0,C 180,E1 -19788.14,E2 -19788.14} C_VEL
LIN {X 0,Y 241.996,Z 503.717,A -85,B 0,C 180,E1 -19790.85,E2 -19790.85} C_VEL
LIN {X 0,Y 244.926,Z 497.403,A -85,B 0,C 180,E1 -19793.41,E2 -19793.41} C_VEL
LIN {X 0,Y 248.473,Z 489.219,A -85,B 0,C 180,E1 -19795.946,E2 -19795.946} C_VEL
LIN {X 0,Y 251.704,Z 480.867,A -85,B 0,C 180,E1 -19798.001,E2 -19798.001} C_VEL
LIN {X 0,Y 255.238,Z 470.593,A -85,B 0,C 180,E1 -19800.001,E2 -19800.001} C_VEL
LIN {X 0,Y 258.523,Z 459.234,A -85,B 0,C 180,E1 -19801.734,E2 -19801.734} C_VEL
LIN {X 0,Y 261.365,Z 447.88,A -85,B 0,C 180,E1 -19803.084,E2 -19803.084} C_VEL
LIN {X 0,Y 264.012,Z 434.489,A -85,B 0,C 180,E1 -19804.294,E2 -19804.294} C_VEL
LIN {X 0,Y 265.865,Z 422.008,A -85,B 0,C 180,E1 -19805.119,E2 -19805.119} C_VEL
LIN {X 0,Y 267.336,Z 407.331,A -85,B 0,C 180,E1 -19805.753,E2 -19805.753} C_VEL
LIN {X 0,Y 271.368,Z 363.024,A -85,B 0,C 180,E1 -19807.357,E2 -19807.357} C_VEL
LIN {X 0,Y 268.589,Z 357.349,A -85,B 0,C 180,E1 -19808.508,E2 -19808.508} C_VEL
LIN {X 0,Y 262.657,Z 347.021,A -85,B 0,C 180,E1 -19811.131,E2 -19811.131} C_VEL
LIN {X 0,Y 259.248,Z 342.04,A -85,B 0,C 180,E1 -19812.787,E2 -19812.787} C_VEL
LIN {X 0,Y 255.927,Z 337.4,A -85,B 0,C 180,E1 -19814.64,E2 -19814.64} C_VEL
LIN {X 0,Y 252.689,Z 333.04,A -85,B 0,C 180,E1 -19816.706,E2 -19816.706} C_VEL
LIN {X 0,Y 251.534,Z 331.817,A -85,B 0,C 180,E1 -19817.512,E2 -19817.512} C_VEL
LIN {X 0,Y 250.289,Z 331.245,A -85,B 0,C 180,E1 -19818.355,E2 -19818.355} C_VEL
LIN {X 0,Y 247.777,Z 331.36,A -85,B 0,C 180,E1 -19820.092,E2 -19820.092} C_VEL
LIN {X 0,Y 244.497,Z 332.154,A -85,B 0,C 180,E1 -19822.82,E2 -19822.82} C_VEL
LIN {X 0,Y 243.692,Z 331.869,A -85,B 0,C 180,E1 -19823.749,E2 -19823.749} C_VEL
LIN {X 0,Y 241.909,Z 330.034,A -85,B 0,C 180,E1 -19827.196,E2 -19827.196} C_VEL
LIN {X 0,Y 241.391,Z 329.678,A -85,B 0,C 180,E1 -19829.667,E2 -19829.667} C_VEL
LIN {X 0,Y 241.83,Z 330.96,A -85,B 0,C 180,E1 -19834.018,E2 -19834.018} C_VEL
LIN {X 0,Y 242.501,Z 332.012,A -85,B 0,C 180,E1 -19835.643,E2 -19835.643} C_VEL
LIN {X 0,Y 245.163,Z 337.006,A -85,B 0,C 180,E1 -19839.772,E2 -19839.772} C_VEL
LIN {X 0,Y 247.498,Z 340.496,A -85,B 0,C 180,E1 -19842.054,E2 -19842.054} C_VEL
LIN {X 0,Y 251.563,Z 347.493,A -85,B 0,C 180,E1 -19845.264,E2 -19845.264} C_VEL
LIN {X 0,Y 254.917,Z 353.764,A -85,B 0,C 180,E1 -19847.419,E2 -19847.419} C_VEL
LIN {X 0,Y 257.911,Z 359.822,A -85,B 0,C 180,E1 -19849.141,E2 -19849.141} C_VEL
LIN {X 0,Y 261.265,Z 367.317,A -85,B 0,C 180,E1 -19850.917,E2 -19850.917} C_VEL
LIN {X 0,Y 263.851,Z 374.46,A -85,B 0,C 180,E1 -19852.227,E2 -19852.227} C_VEL
LIN {X 0,Y 264.697,Z 387.556,A -85,B 0,C 180,E1 -19853.346,E2 -19853.346} C_VEL
LIN {X 0,Y 264.764,Z 392.377,A -85,B 0,C 180,E1 -19853.679,E2 -19853.679} C_VEL
LIN {X 0,Y 260.396,Z 436.557,A -85,B 0,C 180,E1 -19855.322,E2 -19855.322} C_VEL
LIN {X 0,Y 258.157,Z 450.288,A -85,B 0,C 180,E1 -19856.083,E2 -19856.083} C_VEL
LIN {X 0,Y 255.279,Z 463.007,A -85,B 0,C 180,E1 -19857.069,E2 -19857.069} C_VEL
LIN {X 0,Y 252.082,Z 474.581,A -85,B 0,C 180,E1 -19858.255,E2 -19858.255} C_VEL
LIN {X 0,Y 248.266,Z 486.447,A -85,B 0,C 180,E1 -19859.843,E2 -19859.843} C_VEL
LIN {X 0,Y 244.483,Z 497.118,A -85,B 0,C 180,E1 -19861.691,E2 -19861.691} C_VEL
LIN {X 0,Y 240.976,Z 505.959,A -85,B 0,C 180,E1 -19863.598,E2 -19863.598} C_VEL
LIN {X 0,Y 237.306,Z 514.693,A -85,B 0,C 180,E1 -19865.975,E2 -19865.975} C_VEL
LIN {X 0,Y 233.875,Z 522.394,A -85,B 0,C 180,E1 -19868.681,E2 -19868.681} C_VEL
LIN {X 0,Y 231.234,Z 528.433,A -85,B 0,C 180,E1 -19871.394,E2 -19871.394} C_VEL
LIN {X 0,Y 229.067,Z 532.897,A -85,B 0,C 180,E1 -19873.975,E2 -19873.975} C_VEL
LIN {X 0,Y 227.873,Z 535.31,A -85,B 0,C 180,E1 -19875.72,E2 -19875.72} C_VEL
LIN {X 0,Y 227.043,Z 537.252,A -85,B 0,C 180,E1 -19877.49,E2 -19877.49} C_VEL
LIN {X 0,Y 226.035,Z 539.925,A -85,B 0,C 180,E1 -19881.06,E2 -19881.06} C_VEL
LIN {X 0,Y 225.822,Z 540.677,A -85,B 0,C 180,E1 -19882.852,E2 -19882.852} C_VEL
LIN {X 0,Y 225.759,Z 541.008,A -85,B 0,C 180,E1 -19884.998,E2 -19884.998} C_VEL
LIN {X 0,Y 225.909,Z 540.418,A -85,B 0,C 180,E1 -19888.22,E2 -19888.22} C_VEL
LIN {X 0,Y 226.094,Z 539.515,A -85,B 0,C 180,E1 -19890.003,E2 -19890.003} C_VEL
LIN {X 0,Y 225.986,Z 538.124,A -85,B 0,C 180,E1 -19891.785,E2 -19891.785} C_VEL
LIN {X 0,Y 226.084,Z 535.161,A -85,B 0,C 180,E1 -19894.46,E2 -19894.46} C_VEL
LIN {X 0,Y 226.069,Z 531.001,A -85,B 0,C 180,E1 -19897.145,E2 -19897.145} C_VEL
LIN {X 0,Y 226.424,Z 524.531,A -85,B 0,C 180,E1 -19900.283,E2 -19900.283} C_VEL
LIN {X 0,Y 227.124,Z 517.416,A -85,B 0,C 180,E1 -19902.966,E2 -19902.966} C_VEL
LIN {X 0,Y 228.292,Z 508.45,A -85,B 0,C 180,E1 -19905.628,E2 -19905.628} C_VEL
LIN {X 0,Y 229.498,Z 499.231,A -85,B 0,C 180,E1 -19907.833,E2 -19907.833} C_VEL
LIN {X 0,Y 230.964,Z 489.112,A -85,B 0,C 180,E1 -19909.788,E2 -19909.788} C_VEL
LIN {X 0,Y 232.445,Z 477.94,A -85,B 0,C 180,E1 -19911.507,E2 -19911.507} C_VEL
LIN {X 0,Y 233.949,Z 465.644,A -85,B 0,C 180,E1 -19912.988,E2 -19912.988} C_VEL
LIN {X 0,Y 235.303,Z 452.811,A -85,B 0,C 180,E1 -19914.131,E2 -19914.131} C_VEL
LIN {X 0,Y 236.365,Z 439.707,A -85,B 0,C 180,E1 -19914.952,E2 -19914.952} C_VEL
LIN {X 0,Y 238.654,Z 383.982,A -85,B 0,C 180,E1 -19917.152,E2 -19917.152} C_VEL
LIN {X 0,Y 233.797,Z 337.448,A -85,B 0,C 180,E1 -19919.481,E2 -19919.481} C_VEL
LIN {X 0,Y 231.628,Z 330.251,A -85,B 0,C 180,E1 -19919.993,E2 -19919.993} C_VEL
LIN {X 0,Y 229.392,Z 319.112,A -85,B 0,C 180,E1 -19924.185,E2 -19924.185} C_VEL
LIN {X 0,Y 227.931,Z 312.092,A -85,B 0,C 180,E1 -19926.942,E2 -19926.942} C_VEL
LIN {X 0,Y 227.795,Z 312.109,A -85,B 0,C 180,E1 -19930.382,E2 -19930.382} C_VEL
LIN {X 0,Y 227.806,Z 312.106,A -85,B 0,C 180,E1 -19935.198,E2 -19935.198} C_VEL
LIN {X 0,Y 227.795,Z 312.109,A -85,B 0,C 180,E1 -19939.616,E2 -19939.616} C_VEL
LIN {X 0,Y 227.855,Z 312.1,A -85,B 0,C 180,E1 -19944.123,E2 -19944.123} C_VEL
LIN {X 0,Y 227.834,Z 312.103,A -85,B 0,C 180,E1 -19948.371,E2 -19948.371} C_VEL
LIN {X 0,Y 227.846,Z 312.102,A -85,B 0,C 180,E1 -19952.439,E2 -19952.439} C_VEL
LIN {X 0,Y 227.88,Z 312.095,A -85,B 0,C 180,E1 -19956.363,E2 -19956.363} C_VEL
LIN {X 0,Y 227.884,Z 312.096,A -85,B 0,C 180,E1 -19960.168,E2 -19960.168} C_VEL
LIN {X 0,Y 228.005,Z 312.08,A -85,B 0,C 180,E1 -19963.893,E2 -19963.893} C_VEL
LIN {X 0,Y 228.115,Z 312.072,A -85,B 0,C 180,E1 -19969.346,E2 -19969.346} C_VEL
LIN {X 0,Y 228.302,Z 312.044,A -85,B 0,C 180,E1 -19972.926,E2 -19972.926} C_VEL
LIN {X 0,Y 228.533,Z 312.016,A -85,B 0,C 180,E1 -19978.237,E2 -19978.237} C_VEL
LIN {X 0,Y 228.533,Z 312.015,A -85,B 0,C 180,E1 -19981.761,E2 -19981.761} C_VEL
LIN {X 0,Y 228.299,Z 312.046,A -85,B 0,C 180,E1 -19987.072,E2 -19987.072} C_VEL
LIN {X 0,Y 228.128,Z 312.063,A -85,B 0,C 180,E1 -19990.651,E2 -19990.651} C_VEL
LIN {X 0,Y 228.004,Z 312.082,A -85,B 0,C 180,E1 -19996.105,E2 -19996.105} C_VEL
LIN {X 0,Y 227.904,Z 312.097,A -85,B 0,C 180,E1 -20001.718,E2 -20001.718} C_VEL
LIN {X 0,Y 227.931,Z 312.089,A -85,B 0,C 180,E1 -20006.602,E2 -20006.602} C_VEL
LIN {X 0,Y 227.886,Z 312.098,A -85,B 0,C 180,E1 -20010.29,E2 -20010.29} C_VEL
LIN {X 0,Y 227.869,Z 312.101,A -85,B 0,C 180,E1 -20013.721,E2 -20013.721} C_VEL
LIN {X 0,Y 227.836,Z 312.106,A -85,B 0,C 180,E1 -20018.091,E2 -20018.091} C_VEL
LIN {X 0,Y 227.806,Z 312.105,A -85,B 0,C 180,E1 -20022.742,E2 -20022.742} C_VEL
LIN {X 0,Y 227.9,Z 312.094,A -85,B 0,C 180,E1 -20027.28,E2 -20027.28} C_VEL
LIN {X 0,Y 227.867,Z 312.1,A -85,B 0,C 180,E1 -20031.914,E2 -20031.914} C_VEL
LIN {X 0,Y 227.887,Z 312.099,A -85,B 0,C 180,E1 -20036.373,E2 -20036.373} C_VEL
LIN {X 0,Y 227.901,Z 312.094,A -85,B 0,C 180,E1 -20040.435,E2 -20040.435} C_VEL
LIN {X 0,Y 227.926,Z 312.095,A -85,B 0,C 180,E1 -20044.425,E2 -20044.425} C_VEL
LIN {X 0,Y 227.961,Z 312.089,A -85,B 0,C 180,E1 -20048.286,E2 -20048.286} C_VEL
LIN {X 0,Y 228.033,Z 312.08,A -85,B 0,C 180,E1 -20052.824,E2 -20052.824} C_VEL
LIN {X 0,Y 228.074,Z 312.07,A -85,B 0,C 180,E1 -20057.542,E2 -20057.542} C_VEL
LIN {X 0,Y 228.324,Z 312.042,A -85,B 0,C 180,E1 -20061.145,E2 -20061.145} C_VEL
LIN {X 0,Y 228.356,Z 312.039,A -85,B 0,C 180,E1 -20062.927,E2 -20062.927} C_VEL
LIN {X 0,Y 228.553,Z 312.013,A -85,B 0,C 180,E1 -20068.235,E2 -20068.235} C_VEL
LIN {X 0,Y 228.552,Z 312.013,A -85,B 0,C 180,E1 -20071.759,E2 -20071.759} C_VEL
LIN {X 0,Y 228.354,Z 312.04,A -85,B 0,C 180,E1 -20077.068,E2 -20077.068} C_VEL
LIN {X 0,Y 228.166,Z 312.064,A -85,B 0,C 180,E1 -20080.646,E2 -20080.646} C_VEL
LIN {X 0,Y 228.058,Z 312.073,A -85,B 0,C 180,E1 -20086.098,E2 -20086.098} C_VEL
LIN {X 0,Y 227.956,Z 312.089,A -85,B 0,C 180,E1 -20089.819,E2 -20089.819} C_VEL
LIN {X 0,Y 227.918,Z 312.094,A -85,B 0,C 180,E1 -20093.627,E2 -20093.627} C_VEL
LIN {X 0,Y 227.873,Z 312.099,A -85,B 0,C 180,E1 -20097.55,E2 -20097.55} C_VEL
LIN {X 0,Y 227.854,Z 312.103,A -85,B 0,C 180,E1 -20101.618,E2 -20101.618} C_VEL
LIN {X 0,Y 227.88,Z 312.172,A -85,B 0,C 180,E1 -20102.134,E2 -20102.134} C_VEL
LIN {X 0,Y 239.727,Z 343.698,A -85,B 0,C 180,E1 -20104.475,E2 -20104.475} C_VEL
LIN {X 0,Y 236.64,Z 413.395,A -85,B 0,C 180,E1 -20107.179,E2 -20107.179} C_VEL
LIN {X 0,Y 235.922,Z 426.451,A -85,B 0,C 180,E1 -20108.009,E2 -20108.009} C_VEL
LIN {X 0,Y 234.837,Z 438.684,A -85,B 0,C 180,E1 -20109.084,E2 -20109.084} C_VEL
LIN {X 0,Y 233.506,Z 451.067,A -85,B 0,C 180,E1 -20110.54,E2 -20110.54} C_VEL
LIN {X 0,Y 231.949,Z 463.341,A -85,B 0,C 180,E1 -20112.393,E2 -20112.393} C_VEL
LIN {X 0,Y 230.499,Z 474.348,A -85,B 0,C 180,E1 -20114.52,E2 -20114.52} C_VEL
LIN {X 0,Y 229.095,Z 484.475,A -85,B 0,C 180,E1 -20116.958,E2 -20116.958} C_VEL
LIN {X 0,Y 227.893,Z 493.282,A -85,B 0,C 180,E1 -20119.639,E2 -20119.639} C_VEL
LIN {X 0,Y 226.963,Z 500.244,A -85,B 0,C 180,E1 -20122.291,E2 -20122.291} C_VEL
LIN {X 0,Y 226.387,Z 505.793,A -85,B 0,C 180,E1 -20124.949,E2 -20124.949} C_VEL
LIN {X 0,Y 225.886,Z 510.743,A -85,B 0,C 180,E1 -20128.068,E2 -20128.068} C_VEL
LIN {X 0,Y 225.631,Z 513.784,A -85,B 0,C 180,E1 -20130.693,E2 -20130.693} C_VEL
LIN {X 0,Y 225.823,Z 516.335,A -85,B 0,C 180,E1 -20134.171,E2 -20134.171} C_VEL
LIN {X 0,Y 226.115,Z 517.113,A -85,B 0,C 180,E1 -20136.169,E2 -20136.169} C_VEL
LIN {X 0,Y 226.702,Z 517.33,A -85,B 0,C 180,E1 -20138.417,E2 -20138.417} C_VEL
LIN {X 0,Y 227.291,Z 517.09,A -85,B 0,C 180,E1 -20140.116,E2 -20140.116} C_VEL
LIN {X 0,Y 228.401,Z 516.079,A -85,B 0,C 180,E1 -20142.504,E2 -20142.504} C_VEL
LIN {X 0,Y 230.431,Z 513.378,A -85,B 0,C 180,E1 -20145.878,E2 -20145.878} C_VEL
LIN {X 0,Y 232.691,Z 509.782,A -85,B 0,C 180,E1 -20148.679,E2 -20148.679} C_VEL
LIN {X 0,Y 235.409,Z 504.917,A -85,B 0,C 180,E1 -20151.416,E2 -20151.416} C_VEL
LIN {X 0,Y 238.572,Z 498.708,A -85,B 0,C 180,E1 -20154.083,E2 -20154.083} C_VEL
LIN {X 0,Y 242.291,Z 490.804,A -85,B 0,C 180,E1 -20156.675,E2 -20156.675} C_VEL
LIN {X 0,Y 245.985,Z 481.858,A -85,B 0,C 180,E1 -20158.945,E2 -20158.945} C_VEL
LIN {X 0,Y 249.765,Z 471.567,A -85,B 0,C 180,E1 -20161.008,E2 -20161.008} C_VEL
LIN {X 0,Y 253.266,Z 460.371,A -85,B 0,C 180,E1 -20162.765,E2 -20162.765} C_VEL
LIN {X 0,Y 256.264,Z 449.21,A -85,B 0,C 180,E1 -20164.129,E2 -20164.129} C_VEL
LIN {X 0,Y 258.812,Z 437.282,A -85,B 0,C 180,E1 -20165.259,E2 -20165.259} C_VEL
LIN {X 0,Y 261.044,Z 423.344,A -85,B 0,C 180,E1 -20166.227,E2 -20166.227} C_VEL
LIN {X 0,Y 262.617,Z 409.122,A -85,B 0,C 180,E1 -20166.86,E2 -20166.86} C_VEL
LIN {X 0,Y 266.819,Z 365.988,A -85,B 0,C 180,E1 -20168.457,E2 -20168.457} C_VEL
LIN {X 0,Y 262.082,Z 357.198,A -85,B 0,C 180,E1 -20170.566,E2 -20170.566} C_VEL
LIN {X 0,Y 259,Z 351.716,A -85,B 0,C 180,E1 -20172.1,E2 -20172.1} C_VEL
LIN {X 0,Y 256.479,Z 347.966,A -85,B 0,C 180,E1 -20173.428,E2 -20173.428} C_VEL
LIN {X 0,Y 253.469,Z 343.606,A -85,B 0,C 180,E1 -20175.186,E2 -20175.186} C_VEL
LIN {X 0,Y 250.107,Z 338.986,A -85,B 0,C 180,E1 -20177.491,E2 -20177.491} C_VEL
LIN {X 0,Y 247.781,Z 336.283,A -85,B 0,C 180,E1 -20179.33,E2 -20179.33} C_VEL
LIN {X 0,Y 245.408,Z 333.163,A -85,B 0,C 180,E1 -20181.688,E2 -20181.688} C_VEL
LIN {X 0,Y 243.692,Z 331.869,A -85,B 0,C 180,E1 -20183.749,E2 -20183.749} C_VEL
LIN {X 0,Y 242.709,Z 331.757,A -85,B 0,C 180,E1 -20185.123,E2 -20185.123} C_VEL
LIN {X 0,Y 241.156,Z 333.584,A -85,B 0,C 180,E1 -20187.404,E2 -20187.404} C_VEL
LIN {X 0,Y 240.089,Z 336.444,A -85,B 0,C 180,E1 -20190.184,E2 -20190.184} C_VEL
LIN {X 0,Y 240.011,Z 336.949,A -85,B 0,C 180,E1 -20191.133,E2 -20191.133} C_VEL
LIN {X 0,Y 240.948,Z 338.487,A -85,B 0,C 180,E1 -20195.048,E2 -20195.048} C_VEL
LIN {X 0,Y 243.564,Z 343.916,A -85,B 0,C 180,E1 -20199.542,E2 -20199.542} C_VEL
LIN {X 0,Y 245.504,Z 346.954,A -85,B 0,C 180,E1 -20201.537,E2 -20201.537} C_VEL
LIN {X 0,Y 249.287,Z 353.824,A -85,B 0,C 180,E1 -20204.726,E2 -20204.726} C_VEL
LIN {X 0,Y 252.264,Z 359.76,A -85,B 0,C 180,E1 -20206.792,E2 -20206.792} C_VEL
LIN {X 0,Y 255.079,Z 365.835,A -85,B 0,C 180,E1 -20208.552,E2 -20208.552} C_VEL
LIN {X 0,Y 258.618,Z 374.337,A -85,B 0,C 180,E1 -20210.525,E2 -20210.525} C_VEL
LIN {X 0,Y 259.77,Z 378.282,A -85,B 0,C 180,E1 -20211.221,E2 -20211.221} C_VEL
LIN {X 0,Y 260.459,Z 391.382,A -85,B 0,C 180,E1 -20212.343,E2 -20212.343} C_VEL
LIN {X 0,Y 260.193,Z 395.757,A -85,B 0,C 180,E1 -20212.56,E2 -20212.56} C_VEL
LIN {X 0,Y 255.997,Z 435.705,A -85,B 0,C 180,E1 -20214.073,E2 -20214.073} C_VEL
LIN {X 0,Y 253.462,Z 450.213,A -85,B 0,C 180,E1 -20214.883,E2 -20214.883} C_VEL
LIN {X 0,Y 249.966,Z 464.622,A -85,B 0,C 180,E1 -20216.034,E2 -20216.034} C_VEL
LIN {X 0,Y 246.689,Z 475.793,A -85,B 0,C 180,E1 -20217.235,E2 -20217.235} C_VEL
LIN {X 0,Y 242.697,Z 487.296,A -85,B 0,C 180,E1 -20218.834,E2 -20218.834} C_VEL
LIN {X 0,Y 239.142,Z 496.714,A -85,B 0,C 180,E1 -20220.517,E2 -20220.517} C_VEL
LIN {X 0,Y 235.428,Z 505.47,A -85,B 0,C 180,E1 -20222.444,E2 -20222.444} C_VEL
LIN {X 0,Y 232.151,Z 512.85,A -85,B 0,C 180,E1 -20224.45,E2 -20224.45} C_VEL
LIN {X 0,Y 228.609,Z 520.239,A -85,B 0,C 180,E1 -20226.929,E2 -20226.929} C_VEL
LIN {X 0,Y 225.226,Z 527.077,A -85,B 0,C 180,E1 -20229.93,E2 -20229.93} C_VEL
LIN {X 0,Y 222.977,Z 531.701,A -85,B 0,C 180,E1 -20232.581,E2 -20232.581} C_VEL
LIN {X 0,Y 220.99,Z 535.315,A -85,B 0,C 180,E1 -20235.265,E2 -20235.265} C_VEL
LIN {X 0,Y 219.456,Z 538.617,A -85,B 0,C 180,E1 -20238.926,E2 -20238.926} C_VEL
LIN {X 0,Y 218.999,Z 539.68,A -85,B 0,C 180,E1 -20240.77,E2 -20240.77} C_VEL
LIN {X 0,Y 218.769,Z 540.319,A -85,B 0,C 180,E1 -20242.621,E2 -20242.621} C_VEL
LIN {X 0,Y 218.677,Z 540.557,A -85,B 0,C 180,E1 -20245.081,E2 -20245.081} C_VEL
LIN {X 0,Y 218.838,Z 539.832,A -85,B 0,C 180,E1 -20248.163,E2 -20248.163} C_VEL
LIN {X 0,Y 219.02,Z 538.829,A -85,B 0,C 180,E1 -20250.003,E2 -20250.003} C_VEL
LIN {X 0,Y 218.92,Z 537.326,A -85,B 0,C 180,E1 -20251.842,E2 -20251.842} C_VEL
LIN {X 0,Y 219.029,Z 534.224,A -85,B 0,C 180,E1 -20254.604,E2 -20254.604} C_VEL
LIN {X 0,Y 219.038,Z 529.922,A -85,B 0,C 180,E1 -20257.376,E2 -20257.376} C_VEL
LIN {X 0,Y 219.345,Z 524.339,A -85,B 0,C 180,E1 -20260.152,E2 -20260.152} C_VEL
LIN {X 0,Y 220.007,Z 517.294,A -85,B 0,C 180,E1 -20262.923,E2 -20262.923} C_VEL
LIN {X 0,Y 220.971,Z 510.077,A -85,B 0,C 180,E1 -20265.213,E2 -20265.213} C_VEL
LIN {X 0,Y 222.133,Z 501.262,A -85,B 0,C 180,E1 -20267.493,E2 -20267.493} C_VEL
LIN {X 0,Y 223.733,Z 490.441,A -85,B 0,C 180,E1 -20269.742,E2 -20269.742} C_VEL
LIN {X 0,Y 225.196,Z 479.785,A -85,B 0,C 180,E1 -20271.513,E2 -20271.513} C_VEL
LIN {X 0,Y 226.666,Z 468.001,A -85,B 0,C 180,E1 -20273.045,E2 -20273.045} C_VEL
LIN {X 0,Y 228.178,Z 454.969,A -85,B 0,C 180,E1 -20274.328,E2 -20274.328} C_VEL
LIN {X 0,Y 229.302,Z 442.007,A -85,B 0,C 180,E1 -20275.228,E2 -20275.228} C_VEL
LIN {X 0,Y 230.255,Z 422.639,A -85,B 0,C 180,E1 -20276.086,E2 -20276.086} C_VEL
LIN {X 0,Y 231.757,Z 384.353,A -85,B 0,C 180,E1 -20277.622,E2 -20277.622} C_VEL
LIN {X 0,Y 227.149,Z 339.16,A -85,B 0,C 180,E1 -20279.965,E2 -20279.965} C_VEL
LIN {X 0,Y 224.275,Z 329.781,A -85,B 0,C 180,E1 -20280.683,E2 -20280.683} C_VEL
LIN {X 0,Y 222.213,Z 319.444,A -85,B 0,C 180,E1 -20284.7,E2 -20284.7} C_VEL
LIN {X 0,Y 220.864,Z 312.971,A -85,B 0,C 180,E1 -20287.391,E2 -20287.391} C_VEL
LIN {X 0,Y 220.743,Z 312.987,A -85,B 0,C 180,E1 -20291.958,E2 -20291.958} C_VEL
LIN {X 0,Y 220.749,Z 312.983,A -85,B 0,C 180,E1 -20295.538,E2 -20295.538} C_VEL
LIN {X 0,Y 220.777,Z 312.984,A -85,B 0,C 180,E1 -20300.456,E2 -20300.456} C_VEL
LIN {X 0,Y 220.822,Z 312.978,A -85,B 0,C 180,E1 -20302.791,E2 -20302.791} C_VEL
LIN {X 0,Y 220.797,Z 312.982,A -85,B 0,C 180,E1 -20307.24,E2 -20307.24} C_VEL
LIN {X 0,Y 220.795,Z 312.981,A -85,B 0,C 180,E1 -20311.48,E2 -20311.48} C_VEL
LIN {X 0,Y 220.836,Z 312.974,A -85,B 0,C 180,E1 -20315.56,E2 -20315.56} C_VEL
LIN {X 0,Y 220.842,Z 312.976,A -85,B 0,C 180,E1 -20319.508,E2 -20319.508} C_VEL
LIN {X 0,Y 220.965,Z 312.96,A -85,B 0,C 180,E1 -20323.365,E2 -20323.365} C_VEL
LIN {X 0,Y 221.041,Z 312.951,A -85,B 0,C 180,E1 -20329.001,E2 -20329.001} C_VEL
LIN {X 0,Y 221.237,Z 312.924,A -85,B 0,C 180,E1 -20332.699,E2 -20332.699} C_VEL
LIN {X 0,Y 221.491,Z 312.893,A -85,B 0,C 180,E1 -20338.181,E2 -20338.181} C_VEL
LIN {X 0,Y 221.491,Z 312.892,A -85,B 0,C 180,E1 -20341.817,E2 -20341.817} C_VEL
LIN {X 0,Y 221.234,Z 312.927,A -85,B 0,C 180,E1 -20347.299,E2 -20347.299} C_VEL
LIN {X 0,Y 221.049,Z 312.945,A -85,B 0,C 180,E1 -20350.996,E2 -20350.996} C_VEL
LIN {X 0,Y 220.963,Z 312.958,A -85,B 0,C 180,E1 -20356.633,E2 -20356.633} C_VEL
LIN {X 0,Y 220.834,Z 312.974,A -85,B 0,C 180,E1 -20360.491,E2 -20360.491} C_VEL
LIN {X 0,Y 220.848,Z 312.973,A -85,B 0,C 180,E1 -20364.436,E2 -20364.436} C_VEL
LIN {X 0,Y 220.816,Z 312.976,A -85,B 0,C 180,E1 -20368.515,E2 -20368.515} C_VEL
LIN {X 0,Y 220.807,Z 312.978,A -85,B 0,C 180,E1 -20372.757,E2 -20372.757} C_VEL
LIN {X 0,Y 220.803,Z 312.977,A -85,B 0,C 180,E1 -20377.278,E2 -20377.278} C_VEL
LIN {X 0,Y 220.764,Z 312.987,A -85,B 0,C 180,E1 -20381.953,E2 -20381.953} C_VEL
LIN {X 0,Y 220.858,Z 312.971,A -85,B 0,C 180,E1 -20387.044,E2 -20387.044} C_VEL
LIN {X 0,Y 220.851,Z 312.973,A -85,B 0,C 180,E1 -20390.474,E2 -20390.474} C_VEL
LIN {X 0,Y 220.812,Z 312.977,A -85,B 0,C 180,E1 -20395.048,E2 -20395.048} C_VEL
LIN {X 0,Y 220.831,Z 312.974,A -85,B 0,C 180,E1 -20399.389,E2 -20399.389} C_VEL
LIN {X 0,Y 220.892,Z 312.967,A -85,B 0,C 180,E1 -20403.549,E2 -20403.549} C_VEL
LIN {X 0,Y 220.877,Z 312.969,A -85,B 0,C 180,E1 -20407.553,E2 -20407.553} C_VEL
LIN {X 0,Y 220.983,Z 312.959,A -85,B 0,C 180,E1 -20412.57,E2 -20412.57} C_VEL
LIN {X 0,Y 221.012,Z 312.95,A -85,B 0,C 180,E1 -20417.137,E2 -20417.137} C_VEL
LIN {X 0,Y 221.257,Z 312.924,A -85,B 0,C 180,E1 -20420.86,E2 -20420.86} C_VEL
LIN {X 0,Y 221.31,Z 312.918,A -85,B 0,C 180,E1 -20422.7,E2 -20422.7} C_VEL
LIN {X 0,Y 221.511,Z 312.89,A -85,B 0,C 180,E1 -20428.179,E2 -20428.179} C_VEL
LIN {X 0,Y 221.51,Z 312.89,A -85,B 0,C 180,E1 -20431.815,E2 -20431.815} C_VEL
LIN {X 0,Y 221.291,Z 312.919,A -85,B 0,C 180,E1 -20437.295,E2 -20437.295} C_VEL
LIN {X 0,Y 221.111,Z 312.942,A -85,B 0,C 180,E1 -20440.99,E2 -20440.99} C_VEL
LIN {X 0,Y 221.017,Z 312.952,A -85,B 0,C 180,E1 -20446.625,E2 -20446.625} C_VEL
LIN {X 0,Y 220.911,Z 312.968,A -85,B 0,C 180,E1 -20450.479,E2 -20450.479} C_VEL
LIN {X 0,Y 220.864,Z 312.973,A -85,B 0,C 180,E1 -20454.43,E2 -20454.43} C_VEL
LIN {X 0,Y 220.823,Z 312.977,A -85,B 0,C 180,E1 -20458.509,E2 -20458.509} C_VEL
LIN {X 0,Y 220.83,Z 313.025,A -85,B 0,C 180,E1 -20461.534,E2 -20461.534} C_VEL
LIN {X 0,Y 232.904,Z 345.014,A -85,B 0,C 180,E1 -20463.994,E2 -20463.994} C_VEL
LIN {X 0,Y 229.716,Z 413.992,A -85,B 0,C 180,E1 -20466.758,E2 -20466.758} C_VEL
LIN {X 0,Y 229.003,Z 427.273,A -85,B 0,C 180,E1 -20467.638,E2 -20467.638} C_VEL
LIN {X 0,Y 227.902,Z 439.074,A -85,B 0,C 180,E1 -20468.712,E2 -20468.712} C_VEL
LIN {X 0,Y 226.552,Z 451.36,A -85,B 0,C 180,E1 -20470.202,E2 -20470.202} C_VEL
LIN {X 0,Y 225.141,Z 462.1,A -85,B 0,C 180,E1 -20471.852,E2 -20471.852} C_VEL
LIN {X 0,Y 223.808,Z 472.155,A -85,B 0,C 180,E1 -20473.761,E2 -20473.761} C_VEL
LIN {X 0,Y 222.486,Z 481.63,A -85,B 0,C 180,E1 -20475.978,E2 -20475.978} C_VEL
LIN {X 0,Y 221.138,Z 490.893,A -85,B 0,C 180,E1 -20478.674,E2 -20478.674} C_VEL
LIN {X 0,Y 220.094,Z 498.633,A -85,B 0,C 180,E1 -20481.49,E2 -20481.49} C_VEL
LIN {X 0,Y 219.448,Z 504.02,A -85,B 0,C 180,E1 -20483.935,E2 -20483.935} C_VEL
LIN {X 0,Y 218.953,Z 509.213,A -85,B 0,C 180,E1 -20486.931,E2 -20486.931} C_VEL
LIN {X 0,Y 218.574,Z 513.407,A -85,B 0,C 180,E1 -20490.229,E2 -20490.229} C_VEL
LIN {X 0,Y 218.737,Z 516.497,A -85,B 0,C 180,E1 -20494.092,E2 -20494.092} C_VEL
LIN {X 0,Y 219.306,Z 517.675,A -85,B 0,C 180,E1 -20497.385,E2 -20497.385} C_VEL
LIN {X 0,Y 219.935,Z 517.78,A -85,B 0,C 180,E1 -20499.422,E2 -20499.422} C_VEL
LIN {X 0,Y 221.202,Z 517.005,A -85,B 0,C 180,E1 -20502.365,E2 -20502.365} C_VEL
LIN {X 0,Y 222.966,Z 515.064,A -85,B 0,C 180,E1 -20505.395,E2 -20505.395} C_VEL
LIN {X 0,Y 225.167,Z 512.026,A -85,B 0,C 180,E1 -20508.295,E2 -20508.295} C_VEL
LIN {X 0,Y 227.892,Z 507.785,A -85,B 0,C 180,E1 -20511.131,E2 -20511.131} C_VEL
LIN {X 0,Y 231.155,Z 502.188,A -85,B 0,C 180,E1 -20513.892,E2 -20513.892} C_VEL
LIN {X 0,Y 234.811,Z 495.114,A -85,B 0,C 180,E1 -20516.569,E2 -20516.569} C_VEL
LIN {X 0,Y 238.944,Z 486.255,A -85,B 0,C 180,E1 -20519.132,E2 -20519.132} C_VEL
LIN {X 0,Y 242.842,Z 476.914,A -85,B 0,C 180,E1 -20521.245,E2 -20521.245} C_VEL
LIN {X 0,Y 246.508,Z 466.683,A -85,B 0,C 180,E1 -20523.067,E2 -20523.067} C_VEL
LIN {X 0,Y 249.903,Z 455.502,A -85,B 0,C 180,E1 -20524.638,E2 -20524.638} C_VEL
LIN {X 0,Y 253.045,Z 443.175,A -85,B 0,C 180,E1 -20525.979,E2 -20525.979} C_VEL
LIN {X 0,Y 255.513,Z 430.594,A -85,B 0,C 180,E1 -20527.012,E2 -20527.012} C_VEL
LIN {X 0,Y 257.415,Z 417.585,A -85,B 0,C 180,E1 -20527.765,E2 -20527.765} C_VEL
LIN {X 0,Y 262.32,Z 369.244,A -85,B 0,C 180,E1 -20529.608,E2 -20529.608} C_VEL
LIN {X 0,Y 256.681,Z 358.423,A -85,B 0,C 180,E1 -20532.441,E2 -20532.441} C_VEL
LIN {X 0,Y 253.785,Z 353.917,A -85,B 0,C 180,E1 -20534.067,E2 -20534.067} C_VEL
LIN {X 0,Y 251.063,Z 349.821,A -85,B 0,C 180,E1 -20535.75,E2 -20535.75} C_VEL
LIN {X 0,Y 248.076,Z 345.529,A -85,B 0,C 180,E1 -20537.913,E2 -20537.913} C_VEL
LIN {X 0,Y 243.911,Z 340.107,A -85,B 0,C 180,E1 -20541.828,E2 -20541.828} C_VEL
LIN {X 0,Y 240.739,Z 337.169,A -85,B 0,C 180,E1 -20546.834,E2 -20546.834} C_VEL
LIN {X 0,Y 240.06,Z 336.692,A -85,B 0,C 180,E1 -20549.848,E2 -20549.848} C_VEL
LIN {X 0,Y 240.011,Z 336.949,A -85,B 0,C 180,E1 -20551.133,E2 -20551.133} C_VEL
LIN {X 0,Y 240.057,Z 338.051,A -85,B 0,C 180,E1 -20552.519,E2 -20552.519} C_VEL
LIN {X 0,Y 240.084,Z 340.149,A -85,B 0,C 180,E1 -20553.846,E2 -20553.846} C_VEL
LIN {X 0,Y 240.412,Z 345.696,A -85,B 0,C 180,E1 -20556.396,E2 -20556.396} C_VEL
LIN {X 0,Y 241.151,Z 349.141,A -85,B 0,C 180,E1 -20558.121,E2 -20558.121} C_VEL
LIN {X 0,Y 243.573,Z 353.513,A -85,B 0,C 180,E1 -20561.06,E2 -20561.06} C_VEL
LIN {X 0,Y 246.955,Z 360.012,A -85,B 0,C 180,E1 -20564.121,E2 -20564.121} C_VEL
LIN {X 0,Y 249.506,Z 365.46,A -85,B 0,C 180,E1 -20566.062,E2 -20566.062} C_VEL
LIN {X 0,Y 251.974,Z 370.997,A -85,B 0,C 180,E1 -20567.699,E2 -20567.699} C_VEL
LIN {X 0,Y 255.109,Z 379.057,A -85,B 0,C 180,E1 -20569.626,E2 -20569.626} C_VEL
LIN {X 0,Y 255.894,Z 381.808,A -85,B 0,C 180,E1 -20570.129,E2 -20570.129} C_VEL
LIN {X 0,Y 256.258,Z 394.244,A -85,B 0,C 180,E1 -20571.21,E2 -20571.21} C_VEL
LIN {X 0,Y 251.673,Z 435.68,A -85,B 0,C 180,E1 -20572.796,E2 -20572.796} C_VEL
LIN {X 0,Y 249.224,Z 449.36,A -85,B 0,C 180,E1 -20573.569,E2 -20573.569} C_VEL
LIN {X 0,Y 245.805,Z 462.884,A -85,B 0,C 180,E1 -20574.628,E2 -20574.628} C_VEL
LIN {X 0,Y 242.317,Z 474.214,A -85,B 0,C 180,E1 -20575.817,E2 -20575.817} C_VEL
LIN {X 0,Y 238.083,Z 485.866,A -85,B 0,C 180,E1 -20577.41,E2 -20577.41} C_VEL
LIN {X 0,Y 233.917,Z 496.404,A -85,B 0,C 180,E1 -20579.292,E2 -20579.292} C_VEL
LIN {X 0,Y 229.996,Z 505.149,A -85,B 0,C 180,E1 -20581.238,E2 -20581.238} C_VEL
LIN {X 0,Y 226.505,Z 512.455,A -85,B 0,C 180,E1 -20583.268,E2 -20583.268} C_VEL
LIN {X 0,Y 222.685,Z 519.772,A -85,B 0,C 180,E1 -20585.783,E2 -20585.783} C_VEL
LIN {X 0,Y 219.559,Z 525.697,A -85,B 0,C 180,E1 -20588.371,E2 -20588.371} C_VEL
LIN {X 0,Y 216.983,Z 530.564,A -85,B 0,C 180,E1 -20591.106,E2 -20591.106} C_VEL
LIN {X 0,Y 214.779,Z 534.31,A -85,B 0,C 180,E1 -20593.856,E2 -20593.856} C_VEL
LIN {X 0,Y 213.117,Z 537.081,A -85,B 0,C 180,E1 -20596.658,E2 -20596.658} C_VEL
LIN {X 0,Y 212.445,Z 538.45,A -85,B 0,C 180,E1 -20598.556,E2 -20598.556} C_VEL
LIN {X 0,Y 211.693,Z 539.934,A -85,B 0,C 180,E1 -20602.373,E2 -20602.373} C_VEL
LIN {X 0,Y 211.619,Z 540.054,A -85,B 0,C 180,E1 -20605.092,E2 -20605.092} C_VEL
LIN {X 0,Y 211.766,Z 539.213,A -85,B 0,C 180,E1 -20608.101,E2 -20608.101} C_VEL
LIN {X 0,Y 211.948,Z 538.104,A -85,B 0,C 180,E1 -20610.003,E2 -20610.003} C_VEL
LIN {X 0,Y 211.867,Z 535.565,A -85,B 0,C 180,E1 -20612.855,E2 -20612.855} C_VEL
LIN {X 0,Y 211.967,Z 531.627,A -85,B 0,C 180,E1 -20615.904,E2 -20615.904} C_VEL
LIN {X 0,Y 212.058,Z 527.021,A -85,B 0,C 180,E1 -20618.579,E2 -20618.579} C_VEL
LIN {X 0,Y 212.528,Z 520.766,A -85,B 0,C 180,E1 -20621.446,E2 -20621.446} C_VEL
LIN {X 0,Y 213.45,Z 512.924,A -85,B 0,C 180,E1 -20624.298,E2 -20624.298} C_VEL
LIN {X 0,Y 214.56,Z 504.848,A -85,B 0,C 180,E1 -20626.657,E2 -20626.657} C_VEL
LIN {X 0,Y 216.004,Z 495.011,A -85,B 0,C 180,E1 -20628.989,E2 -20628.989} C_VEL
LIN {X 0,Y 217.612,Z 484.142,A -85,B 0,C 180,E1 -20631.058,E2 -20631.058} C_VEL
LIN {X 0,Y 219.214,Z 471.881,A -85,B 0,C 180,E1 -20632.876,E2 -20632.876} C_VEL
LIN {X 0,Y 220.793,Z 459.127,A -85,B 0,C 180,E1 -20634.319,E2 -20634.319} C_VEL
LIN {X 0,Y 222.16,Z 444.805,A -85,B 0,C 180,E1 -20635.47,E2 -20635.47} C_VEL
LIN {X 0,Y 222.895,Z 431.101,A -85,B 0,C 180,E1 -20636.195,E2 -20636.195} C_VEL
LIN {X 0,Y 224.974,Z 385.065,A -85,B 0,C 180,E1 -20638.096,E2 -20638.096} C_VEL
LIN {X 0,Y 220.563,Z 341.093,A -85,B 0,C 180,E1 -20640.446,E2 -20640.446} C_VEL
LIN {X 0,Y 216.993,Z 329.521,A -85,B 0,C 180,E1 -20641.305,E2 -20641.305} C_VEL
LIN {X 0,Y 214.907,Z 319.077,A -85,B 0,C 180,E1 -20645.529,E2 -20645.529} C_VEL
LIN {X 0,Y 213.817,Z 313.848,A -85,B 0,C 180,E1 -20647.752,E2 -20647.752} C_VEL
LIN {X 0,Y 213.695,Z 313.867,A -85,B 0,C 180,E1 -20651.128,E2 -20651.128} C_VEL
LIN {X 0,Y 213.7,Z 313.864,A -85,B 0,C 180,E1 -20653.679,E2 -20653.679} C_VEL
LIN {X 0,Y 213.699,Z 313.861,A -85,B 0,C 180,E1 -20656.344,E2 -20656.344} C_VEL
LIN {X 0,Y 213.699,Z 313.865,A -85,B 0,C 180,E1 -20661.327,E2 -20661.327} C_VEL
LIN {X 0,Y 213.742,Z 313.858,A -85,B 0,C 180,E1 -20666.014,E2 -20666.014} C_VEL
LIN {X 0,Y 213.735,Z 313.859,A -85,B 0,C 180,E1 -20670.446,E2 -20670.446} C_VEL
LIN {X 0,Y 213.772,Z 313.856,A -85,B 0,C 180,E1 -20674.697,E2 -20674.697} C_VEL
LIN {X 0,Y 213.769,Z 313.854,A -85,B 0,C 180,E1 -20678.798,E2 -20678.798} C_VEL
LIN {X 0,Y 213.874,Z 313.843,A -85,B 0,C 180,E1 -20682.797,E2 -20682.797} C_VEL
LIN {X 0,Y 213.909,Z 313.836,A -85,B 0,C 180,E1 -20686.703,E2 -20686.703} C_VEL
LIN {X 0,Y 214.115,Z 313.812,A -85,B 0,C 180,E1 -20690.553,E2 -20690.553} C_VEL
LIN {X 0,Y 214.075,Z 313.814,A -85,B 0,C 180,E1 -20694.347,E2 -20694.347} C_VEL
LIN {X 0,Y 214.424,Z 313.774,A -85,B 0,C 180,E1 -20698.121,E2 -20698.121} C_VEL
LIN {X 0,Y 214.522,Z 313.761,A -85,B 0,C 180,E1 -20699.999,E2 -20699.999} C_VEL
LIN {X 0,Y 214.424,Z 313.771,A -85,B 0,C 180,E1 -20701.877,E2 -20701.877} C_VEL
LIN {X 0,Y 214.173,Z 313.808,A -85,B 0,C 180,E1 -20707.541,E2 -20707.541} C_VEL
LIN {X 0,Y 213.979,Z 313.827,A -85,B 0,C 180,E1 -20711.364,E2 -20711.364} C_VEL
LIN {X 0,Y 213.869,Z 313.844,A -85,B 0,C 180,E1 -20715.241,E2 -20715.241} C_VEL
LIN {X 0,Y 213.779,Z 313.851,A -85,B 0,C 180,E1 -20719.192,E2 -20719.192} C_VEL
LIN {X 0,Y 213.786,Z 313.854,A -85,B 0,C 180,E1 -20723.233,E2 -20723.233} C_VEL
LIN {X 0,Y 213.821,Z 313.847,A -85,B 0,C 180,E1 -20727.45,E2 -20727.45} C_VEL
LIN {X 0,Y 213.759,Z 313.859,A -85,B 0,C 180,E1 -20731.738,E2 -20731.738} C_VEL
LIN {X 0,Y 213.736,Z 313.859,A -85,B 0,C 180,E1 -20736.289,E2 -20736.289} C_VEL
LIN {X 0,Y 213.706,Z 313.863,A -85,B 0,C 180,E1 -20741.125,E2 -20741.125} C_VEL
LIN {X 0,Y 213.775,Z 313.856,A -85,B 0,C 180,E1 -20746.34,E2 -20746.34} C_VEL
LIN {X 0,Y 213.789,Z 313.852,A -85,B 0,C 180,E1 -20749.119,E2 -20749.119} C_VEL
LIN {X 0,Y 213.75,Z 313.855,A -85,B 0,C 180,E1 -20753.714,E2 -20753.714} C_VEL
LIN {X 0,Y 213.767,Z 313.858,A -85,B 0,C 180,E1 -20758.262,E2 -20758.262} C_VEL
LIN {X 0,Y 213.824,Z 313.849,A -85,B 0,C 180,E1 -20762.603,E2 -20762.603} C_VEL
LIN {X 0,Y 213.851,Z 313.845,A -85,B 0,C 180,E1 -20766.952,E2 -20766.952} C_VEL
LIN {X 0,Y 213.942,Z 313.835,A -85,B 0,C 180,E1 -20772.802,E2 -20772.802} C_VEL
LIN {X 0,Y 213.953,Z 313.831,A -85,B 0,C 180,E1 -20776.705,E2 -20776.705} C_VEL
LIN {X 0,Y 214.195,Z 313.805,A -85,B 0,C 180,E1 -20780.556,E2 -20780.556} C_VEL
LIN {X 0,Y 214.246,Z 313.799,A -85,B 0,C 180,E1 -20782.458,E2 -20782.458} C_VEL
LIN {X 0,Y 214.444,Z 313.77,A -85,B 0,C 180,E1 -20788.119,E2 -20788.119} C_VEL
LIN {X 0,Y 214.548,Z 313.758,A -85,B 0,C 180,E1 -20789.997,E2 -20789.997} C_VEL
LIN {X 0,Y 214.443,Z 313.771,A -85,B 0,C 180,E1 -20791.875,E2 -20791.875} C_VEL
LIN {X 0,Y 214.231,Z 313.798,A -85,B 0,C 180,E1 -20797.536,E2 -20797.536} C_VEL
LIN {X 0,Y 214.042,Z 313.821,A -85,B 0,C 180,E1 -20801.358,E2 -20801.358} C_VEL
LIN {X 0,Y 213.931,Z 313.834,A -85,B 0,C 180,E1 -20805.232,E2 -20805.232} C_VEL
LIN {X 0,Y 213.873,Z 313.846,A -85,B 0,C 180,E1 -20809.179,E2 -20809.179} C_VEL
LIN {X 0,Y 213.849,Z 313.848,A -85,B 0,C 180,E1 -20813.221,E2 -20813.221} C_VEL
LIN {X 0,Y 213.817,Z 313.851,A -85,B 0,C 180,E1 -20817.445,E2 -20817.445} C_VEL
LIN {X 0,Y 213.787,Z 313.856,A -85,B 0,C 180,E1 -20820.898,E2 -20820.898} C_VEL
LIN {X 0,Y 226.198,Z 346.993,A -85,B 0,C 180,E1 -20823.537,E2 -20823.537} C_VEL
LIN {X 0,Y 222.856,Z 413.95,A -85,B 0,C 180,E1 -20826.309,E2 -20826.309} C_VEL
LIN {X 0,Y 222.077,Z 427.842,A -85,B 0,C 180,E1 -20827.26,E2 -20827.26} C_VEL
LIN {X 0,Y 220.81,Z 440.79,A -85,B 0,C 180,E1 -20828.504,E2 -20828.504} C_VEL
LIN {X 0,Y 219.381,Z 453.262,A -85,B 0,C 180,E1 -20830.108,E2 -20830.108} C_VEL
LIN {X 0,Y 217.749,Z 465.158,A -85,B 0,C 180,E1 -20832.07,E2 -20832.07} C_VEL
LIN {X 0,Y 216.237,Z 476.065,A -85,B 0,C 180,E1 -20834.356,E2 -20834.356} C_VEL
LIN {X 0,Y 214.979,Z 484.93,A -85,B 0,C 180,E1 -20836.646,E2 -20836.646} C_VEL
LIN {X 0,Y 213.839,Z 492.688,A -85,B 0,C 180,E1 -20839.094,E2 -20839.094} C_VEL
LIN {X 0,Y 212.851,Z 499.833,A -85,B 0,C 180,E1 -20841.884,E2 -20841.884} C_VEL
LIN {X 0,Y 212.239,Z 505.4,A -85,B 0,C 180,E1 -20844.587,E2 -20844.587} C_VEL
LIN {X 0,Y 211.736,Z 510.714,A -85,B 0,C 180,E1 -20847.923,E2 -20847.923} C_VEL
LIN {X 0,Y 211.432,Z 514.451,A -85,B 0,C 180,E1 -20851.186,E2 -20851.186} C_VEL
LIN {X 0,Y 211.672,Z 516.857,A -85,B 0,C 180,E1 -20854.43,E2 -20854.43} C_VEL
LIN {X 0,Y 212.34,Z 518.112,A -85,B 0,C 180,E1 -20857.91,E2 -20857.91} C_VEL
LIN {X 0,Y 213.34,Z 518.134,A -85,B 0,C 180,E1 -20860.767,E2 -20860.767} C_VEL
LIN {X 0,Y 214.34,Z 517.568,A -85,B 0,C 180,E1 -20862.837,E2 -20862.837} C_VEL
LIN {X 0,Y 215.514,Z 516.532,A -85,B 0,C 180,E1 -20864.878,E2 -20864.878} C_VEL
LIN {X 0,Y 217.683,Z 514.036,A -85,B 0,C 180,E1 -20867.887,E2 -20867.887} C_VEL
LIN {X 0,Y 220.543,Z 510.093,A -85,B 0,C 180,E1 -20871.011,E2 -20871.011} C_VEL
LIN {X 0,Y 223.618,Z 505.405,A -85,B 0,C 180,E1 -20873.686,E2 -20873.686} C_VEL
LIN {X 0,Y 227.311,Z 499.112,A -85,B 0,C 180,E1 -20876.456,E2 -20876.456} C_VEL
LIN {X 0,Y 231.249,Z 491.683,A -85,B 0,C 180,E1 -20878.958,E2 -20878.958} C_VEL
LIN {X 0,Y 235.45,Z 482.766,A -85,B 0,C 180,E1 -20881.284,E2 -20881.284} C_VEL
LIN {X 0,Y 239.583,Z 472.697,A -85,B 0,C 180,E1 -20883.364,E2 -20883.364} C_VEL
LIN {X 0,Y 243.582,Z 461.401,A -85,B 0,C 180,E1 -20885.174,E2 -20885.174} C_VEL
LIN {X 0,Y 246.848,Z 450.491,A -85,B 0,C 180,E1 -20886.54,E2 -20886.54} C_VEL
LIN {X 0,Y 249.724,Z 438.559,A -85,B 0,C 180,E1 -20887.697,E2 -20887.697} C_VEL
LIN {X 0,Y 252.118,Z 425.344,A -85,B 0,C 180,E1 -20888.646,E2 -20888.646} C_VEL
LIN {X 0,Y 253.781,Z 412.459,A -85,B 0,C 180,E1 -20889.267,E2 -20889.267} C_VEL
LIN {X 0,Y 258.115,Z 372.786,A -85,B 0,C 180,E1 -20890.77,E2 -20890.77} C_VEL
LIN {X 0,Y 253.563,Z 363.748,A -85,B 0,C 180,E1 -20893.263,E2 -20893.263} C_VEL
LIN {X 0,Y 249.417,Z 356.949,A -85,B 0,C 180,E1 -20895.857,E2 -20895.857} C_VEL
LIN {X 0,Y 245.91,Z 351.901,A -85,B 0,C 180,E1 -20898.475,E2 -20898.475} C_VEL
LIN {X 0,Y 242.269,Z 346.861,A -85,B 0,C 180,E1 -20902.156,E2 -20902.156} C_VEL
LIN {X 0,Y 239.336,Z 344.075,A -85,B 0,C 180,E1 -20907.004,E2 -20907.004} C_VEL
LIN {X 0,Y 238.702,Z 343.708,A -85,B 0,C 180,E1 -20910.035,E2 -20910.035} C_VEL
LIN {X 0,Y 239.351,Z 345.116,A -85,B 0,C 180,E1 -20914.419,E2 -20914.419} C_VEL
LIN {X 0,Y 241.151,Z 349.141,A -85,B 0,C 180,E1 -20918.121,E2 -20918.121} C_VEL
LIN {X 0,Y 241.844,Z 351.927,A -85,B 0,C 180,E1 -20919.352,E2 -20919.352} C_VEL
LIN {X 0,Y 244.067,Z 364.634,A -85,B 0,C 180,E1 -20922.944,E2 -20922.944} C_VEL
LIN {X 0,Y 245.354,Z 367.741,A -85,B 0,C 180,E1 -20924.098,E2 -20924.098} C_VEL
LIN {X 0,Y 248.285,Z 374.424,A -85,B 0,C 180,E1 -20926.358,E2 -20926.358} C_VEL
LIN {X 0,Y 251.414,Z 382.999,A -85,B 0,C 180,E1 -20928.539,E2 -20928.539} C_VEL
LIN {X 0,Y 252.118,Z 385.37,A -85,B 0,C 180,E1 -20929.015,E2 -20929.015} C_VEL
LIN {X 0,Y 252.266,Z 395.94,A -85,B 0,C 180,E1 -20929.923,E2 -20929.923} C_VEL
LIN {X 0,Y 247.622,Z 435.162,A -85,B 0,C 180,E1 -20931.435,E2 -20931.435} C_VEL
LIN {X 0,Y 245.095,Z 448.64,A -85,B 0,C 180,E1 -20932.207,E2 -20932.207} C_VEL
LIN {X 0,Y 241.786,Z 461.249,A -85,B 0,C 180,E1 -20933.173,E2 -20933.173} C_VEL
LIN {X 0,Y 237.637,Z 474.292,A -85,B 0,C 180,E1 -20934.529,E2 -20934.529} C_VEL
LIN {X 0,Y 233.232,Z 485.824,A -85,B 0,C 180,E1 -20936.127,E2 -20936.127} C_VEL
LIN {X 0,Y 228.808,Z 496.216,A -85,B 0,C 180,E1 -20938.012,E2 -20938.012} C_VEL
LIN {X 0,Y 224.679,Z 504.833,A -85,B 0,C 180,E1 -20939.975,E2 -20939.975} C_VEL
LIN {X 0,Y 220.842,Z 512.147,A -85,B 0,C 180,E1 -20942.011,E2 -20942.011} C_VEL
LIN {X 0,Y 216.905,Z 519.425,A -85,B 0,C 180,E1 -20944.582,E2 -20944.582} C_VEL
LIN {X 0,Y 213.748,Z 524.883,A -85,B 0,C 180,E1 -20947.021,E2 -20947.021} C_VEL
LIN {X 0,Y 211.097,Z 529.36,A -85,B 0,C 180,E1 -20949.544,E2 -20949.544} C_VEL
LIN {X 0,Y 208.681,Z 533.276,A -85,B 0,C 180,E1 -20952.361,E2 -20952.361} C_VEL
LIN {X 0,Y 207.287,Z 535.356,A -85,B 0,C 180,E1 -20954.267,E2 -20954.267} C_VEL
LIN {X 0,Y 206.178,Z 537,A -85,B 0,C 180,E1 -20956.2,E2 -20956.2} C_VEL
LIN {X 0,Y 204.938,Z 539.08,A -85,B 0,C 180,E1 -20960.131,E2 -20960.131} C_VEL
LIN {X 0,Y 204.557,Z 539.64,A -85,B 0,C 180,E1 -20964.088,E2 -20964.088} C_VEL
LIN {X 0,Y 204.59,Z 539.291,A -85,B 0,C 180,E1 -20966.064,E2 -20966.064} C_VEL
LIN {X 0,Y 204.696,Z 538.528,A -85,B 0,C 180,E1 -20968.036,E2 -20968.036} C_VEL
LIN {X 0,Y 204.879,Z 537.355,A -85,B 0,C 180,E1 -20970.003,E2 -20970.003} C_VEL
LIN {X 0,Y 204.814,Z 534.68,A -85,B 0,C 180,E1 -20972.953,E2 -20972.953} C_VEL
LIN {X 0,Y 204.904,Z 530.888,A -85,B 0,C 180,E1 -20975.909,E2 -20975.909} C_VEL
LIN {X 0,Y 205.045,Z 525.82,A -85,B 0,C 180,E1 -20978.875,E2 -20978.875} C_VEL
LIN {X 0,Y 205.562,Z 519.365,A -85,B 0,C 180,E1 -20981.839,E2 -20981.839} C_VEL
LIN {X 0,Y 206.565,Z 511.212,A -85,B 0,C 180,E1 -20984.786,E2 -20984.786} C_VEL
LIN {X 0,Y 207.711,Z 502.867,A -85,B 0,C 180,E1 -20987.223,E2 -20987.223} C_VEL
LIN {X 0,Y 209.267,Z 492.715,A -85,B 0,C 180,E1 -20989.625,E2 -20989.625} C_VEL
LIN {X 0,Y 210.941,Z 481.278,A -85,B 0,C 180,E1 -20991.757,E2 -20991.757} C_VEL
LIN {X 0,Y 212.445,Z 470.22,A -85,B 0,C 180,E1 -20993.39,E2 -20993.39} C_VEL
LIN {X 0,Y 213.916,Z 458.147,A -85,B 0,C 180,E1 -20994.765,E2 -20994.765} C_VEL
LIN {X 0,Y 215.266,Z 444.469,A -85,B 0,C 180,E1 -20995.892,E2 -20995.892} C_VEL
LIN {X 0,Y 216.01,Z 430.824,A -85,B 0,C 180,E1 -20996.64,E2 -20996.64} C_VEL
LIN {X 0,Y 218.153,Z 385.834,A -85,B 0,C 180,E1 -20998.57,E2 -20998.57} C_VEL
LIN {X 0,Y 213.855,Z 342.736,A -85,B 0,C 180,E1 -21000.957,E2 -21000.957} C_VEL
LIN {X 0,Y 209.701,Z 329.125,A -85,B 0,C 180,E1 -21002.02,E2 -21002.02} C_VEL
LIN {X 0,Y 207.501,Z 318.276,A -85,B 0,C 180,E1 -21006.578,E2 -21006.578} C_VEL
LIN {X 0,Y 206.756,Z 314.728,A -85,B 0,C 180,E1 -21008.139,E2 -21008.139} C_VEL
LIN {X 0,Y 206.617,Z 314.75,A -85,B 0,C 180,E1 -21012.865,E2 -21012.865} C_VEL
LIN {X 0,Y 206.616,Z 314.746,A -85,B 0,C 180,E1 -21017.132,E2 -21017.132} C_VEL
LIN {X 0,Y 206.668,Z 314.74,A -85,B 0,C 180,E1 -21021.455,E2 -21021.455} C_VEL
LIN {X 0,Y 206.697,Z 314.737,A -85,B 0,C 180,E1 -21024.687,E2 -21024.687} C_VEL
LIN {X 0,Y 206.686,Z 314.739,A -85,B 0,C 180,E1 -21029.332,E2 -21029.332} C_VEL
LIN {X 0,Y 206.696,Z 314.736,A -85,B 0,C 180,E1 -21033.766,E2 -21033.766} C_VEL
LIN {X 0,Y 206.708,Z 314.732,A -85,B 0,C 180,E1 -21038.037,E2 -21038.037} C_VEL
LIN {X 0,Y 206.796,Z 314.723,A -85,B 0,C 180,E1 -21042.189,E2 -21042.189} C_VEL
LIN {X 0,Y 206.851,Z 314.714,A -85,B 0,C 180,E1 -21046.24,E2 -21046.24} C_VEL
LIN {X 0,Y 207.063,Z 314.69,A -85,B 0,C 180,E1 -21050.228,E2 -21050.228} C_VEL
LIN {X 0,Y 207.037,Z 314.691,A -85,B 0,C 180,E1 -21054.154,E2 -21054.154} C_VEL
LIN {X 0,Y 207.361,Z 314.654,A -85,B 0,C 180,E1 -21058.057,E2 -21058.057} C_VEL
LIN {X 0,Y 207.489,Z 314.637,A -85,B 0,C 180,E1 -21059.999,E2 -21059.999} C_VEL
LIN {X 0,Y 207.361,Z 314.651,A -85,B 0,C 180,E1 -21061.941,E2 -21061.941} C_VEL
LIN {X 0,Y 207.116,Z 314.685,A -85,B 0,C 180,E1 -21067.8,E2 -21067.8} C_VEL
LIN {X 0,Y 206.9,Z 314.712,A -85,B 0,C 180,E1 -21071.759,E2 -21071.759} C_VEL
LIN {X 0,Y 206.801,Z 314.726,A -85,B 0,C 180,E1 -21075.775,E2 -21075.775} C_VEL
LIN {X 0,Y 206.7,Z 314.736,A -85,B 0,C 180,E1 -21079.876,E2 -21079.876} C_VEL
LIN {X 0,Y 206.73,Z 314.733,A -85,B 0,C 180,E1 -21084.075,E2 -21084.075} C_VEL
LIN {X 0,Y 206.728,Z 314.731,A -85,B 0,C 180,E1 -21088.42,E2 -21088.42} C_VEL
LIN {X 0,Y 206.691,Z 314.736,A -85,B 0,C 180,E1 -21092.958,E2 -21092.958} C_VEL
LIN {X 0,Y 206.673,Z 314.739,A -85,B 0,C 180,E1 -21097.74,E2 -21097.74} C_VEL
LIN {X 0,Y 206.636,Z 314.745,A -85,B 0,C 180,E1 -21101.563,E2 -21101.563} C_VEL
LIN {X 0,Y 206.676,Z 314.737,A -85,B 0,C 180,E1 -21105.568,E2 -21105.568} C_VEL
LIN {X 0,Y 206.72,Z 314.735,A -85,B 0,C 180,E1 -21109.763,E2 -21109.763} C_VEL
LIN {X 0,Y 206.721,Z 314.732,A -85,B 0,C 180,E1 -21112.27,E2 -21112.27} C_VEL
LIN {X 0,Y 206.703,Z 314.735,A -85,B 0,C 180,E1 -21117.043,E2 -21117.043} C_VEL
LIN {X 0,Y 206.762,Z 314.727,A -85,B 0,C 180,E1 -21122.097,E2 -21122.097} C_VEL
LIN {X 0,Y 206.784,Z 314.727,A -85,B 0,C 180,E1 -21126.583,E2 -21126.583} C_VEL
LIN {X 0,Y 206.872,Z 314.715,A -85,B 0,C 180,E1 -21132.195,E2 -21132.195} C_VEL
LIN {X 0,Y 206.895,Z 314.713,A -85,B 0,C 180,E1 -21136.243,E2 -21136.243} C_VEL
LIN {X 0,Y 207.132,Z 314.682,A -85,B 0,C 180,E1 -21140.23,E2 -21140.23} C_VEL
LIN {X 0,Y 207.187,Z 314.677,A -85,B 0,C 180,E1 -21142.199,E2 -21142.199} C_VEL
LIN {X 0,Y 207.38,Z 314.65,A -85,B 0,C 180,E1 -21148.055,E2 -21148.055} C_VEL
LIN {X 0,Y 207.513,Z 314.635,A -85,B 0,C 180,E1 -21149.997,E2 -21149.997} C_VEL
LIN {X 0,Y 207.38,Z 314.651,A -85,B 0,C 180,E1 -21151.939,E2 -21151.939} C_VEL
LIN {X 0,Y 207.174,Z 314.677,A -85,B 0,C 180,E1 -21157.795,E2 -21157.795} C_VEL
LIN {X 0,Y 206.978,Z 314.7,A -85,B 0,C 180,E1 -21161.751,E2 -21161.751} C_VEL
LIN {X 0,Y 206.87,Z 314.712,A -85,B 0,C 180,E1 -21165.766,E2 -21165.766} C_VEL
LIN {X 0,Y 206.811,Z 314.724,A -85,B 0,C 180,E1 -21169.861,E2 -21169.861} C_VEL
LIN {X 0,Y 206.759,Z 314.729,A -85,B 0,C 180,E1 -21174.067,E2 -21174.067} C_VEL
LIN {X 0,Y 206.725,Z 314.733,A -85,B 0,C 180,E1 -21178.415,E2 -21178.415} C_VEL
LIN {X 0,Y 206.741,Z 314.732,A -85,B 0,C 180,E1 -21180.227,E2 -21180.227} C_VEL
LIN {X 0,Y 219.273,Z 347.918,A -85,B 0,C 180,E1 -21183.009,E2 -21183.009} C_VEL
LIN {X 0,Y 215.95,Z 414.612,A -85,B 0,C 180,E1 -21185.881,E2 -21185.881} C_VEL
LIN {X 0,Y 215.159,Z 428.221,A -85,B 0,C 180,E1 -21186.845,E2 -21186.845} C_VEL
LIN {X 0,Y 213.881,Z 441.005,A -85,B 0,C 180,E1 -21188.109,E2 -21188.109} C_VEL
LIN {X 0,Y 212.426,Z 453.388,A -85,B 0,C 180,E1 -21189.744,E2 -21189.744} C_VEL
LIN {X 0,Y 210.89,Z 464.372,A -85,B 0,C 180,E1 -21191.579,E2 -21191.579} C_VEL
LIN {X 0,Y 209.39,Z 474.975,A -85,B 0,C 180,E1 -21193.812,E2 -21193.812} C_VEL
LIN {X 0,Y 207.907,Z 485.121,A -85,B 0,C 180,E1 -21196.47,E2 -21196.47} C_VEL
LIN {X 0,Y 206.74,Z 492.928,A -85,B 0,C 180,E1 -21199.007,E2 -21199.007} C_VEL
LIN {X 0,Y 205.702,Z 500.431,A -85,B 0,C 180,E1 -21202.05,E2 -21202.05} C_VEL
LIN {X 0,Y 205.002,Z 506.829,A -85,B 0,C 180,E1 -21205.35,E2 -21205.35} C_VEL
LIN {X 0,Y 204.492,Z 512.063,A -85,B 0,C 180,E1 -21208.969,E2 -21208.969} C_VEL
LIN {X 0,Y 204.333,Z 514.502,A -85,B 0,C 180,E1 -21211.216,E2 -21211.216} C_VEL
LIN {X 0,Y 204.457,Z 516.358,A -85,B 0,C 180,E1 -21213.459,E2 -21213.459} C_VEL
LIN {X 0,Y 204.752,Z 517.653,A -85,B 0,C 180,E1 -21215.677,E2 -21215.677} C_VEL
LIN {X 0,Y 205.236,Z 518.449,A -85,B 0,C 180,E1 -21217.873,E2 -21217.873} C_VEL
LIN {X 0,Y 205.928,Z 518.696,A -85,B 0,C 180,E1 -21220.046,E2 -21220.046} C_VEL
LIN {X 0,Y 206.859,Z 518.485,A -85,B 0,C 180,E1 -21222.196,E2 -21222.196} C_VEL
LIN {X 0,Y 208.028,Z 517.78,A -85,B 0,C 180,E1 -21224.321,E2 -21224.321} C_VEL
LIN {X 0,Y 209.499,Z 516.46,A -85,B 0,C 180,E1 -21226.581,E2 -21226.581} C_VEL
LIN {X 0,Y 211.865,Z 513.857,A -85,B 0,C 180,E1 -21229.489,E2 -21229.489} C_VEL
LIN {X 0,Y 214.907,Z 509.983,A -85,B 0,C 180,E1 -21232.485,E2 -21232.485} C_VEL
LIN {X 0,Y 218.535,Z 504.778,A -85,B 0,C 180,E1 -21235.41,E2 -21235.41} C_VEL
LIN {X 0,Y 222.558,Z 498.171,A -85,B 0,C 180,E1 -21238.191,E2 -21238.191} C_VEL
LIN {X 0,Y 227.175,Z 489.778,A -85,B 0,C 180,E1 -21240.887,E2 -21240.887} C_VEL
LIN {X 0,Y 231.448,Z 481.114,A -85,B 0,C 180,E1 -21243.047,E2 -21243.047} C_VEL
LIN {X 0,Y 235.459,Z 471.566,A -85,B 0,C 180,E1 -21244.949,E2 -21244.949} C_VEL
LIN {X 0,Y 239.638,Z 460.067,A -85,B 0,C 180,E1 -21246.738,E2 -21246.738} C_VEL
LIN {X 0,Y 243.087,Z 448.635,A -85,B 0,C 180,E1 -21248.107,E2 -21248.107} C_VEL
LIN {X 0,Y 246.337,Z 435.196,A -85,B 0,C 180,E1 -21249.339,E2 -21249.339} C_VEL
LIN {X 0,Y 248.736,Z 421.443,A -85,B 0,C 180,E1 -21250.224,E2 -21250.224} C_VEL
LIN {X 0,Y 252.192,Z 391.951,A -85,B 0,C 180,E1 -21251.414,E2 -21251.414} C_VEL
LIN {X 0,Y 253.988,Z 376.284,A -85,B 0,C 180,E1 -21252.007,E2 -21252.007} C_VEL
LIN {X 0,Y 250.622,Z 369.329,A -85,B 0,C 180,E1 -21254.042,E2 -21254.042} C_VEL
LIN {X 0,Y 247.07,Z 363.156,A -85,B 0,C 180,E1 -21256.445,E2 -21256.445} C_VEL
LIN {X 0,Y 243.786,Z 358.191,A -85,B 0,C 180,E1 -21259.09,E2 -21259.09} C_VEL
LIN {X 0,Y 240.609,Z 353.703,A -85,B 0,C 180,E1 -21262.497,E2 -21262.497} C_VEL
LIN {X 0,Y 237.931,Z 351.001,A -85,B 0,C 180,E1 -21267.176,E2 -21267.176} C_VEL
LIN {X 0,Y 237.348,Z 350.722,A -85,B 0,C 180,E1 -21270.225,E2 -21270.225} C_VEL
LIN {X 0,Y 237.993,Z 352.123,A -85,B 0,C 180,E1 -21274.387,E2 -21274.387} C_VEL
LIN {X 0,Y 240.093,Z 357.147,A -85,B 0,C 180,E1 -21278.644,E2 -21278.644} C_VEL
LIN {X 0,Y 241.608,Z 359.936,A -85,B 0,C 180,E1 -21280.52,E2 -21280.52} C_VEL
LIN {X 0,Y 244.552,Z 365.994,A -85,B 0,C 180,E1 -21283.425,E2 -21283.425} C_VEL
LIN {X 0,Y 245.354,Z 367.741,A -85,B 0,C 180,E1 -21284.098,E2 -21284.098} C_VEL
LIN {X 0,Y 246.099,Z 370.146,A -85,B 0,C 180,E1 -21284.791,E2 -21284.791} C_VEL
LIN {X 0,Y 246.404,Z 373.417,A -85,B 0,C 180,E1 -21285.317,E2 -21285.317} C_VEL
LIN {X 0,Y 246.7,Z 381.941,A -85,B 0,C 180,E1 -21286.346,E2 -21286.346} C_VEL
LIN {X 0,Y 247.302,Z 385.105,A -85,B 0,C 180,E1 -21286.932,E2 -21286.932} C_VEL
LIN {X 0,Y 248.565,Z 389.264,A -85,B 0,C 180,E1 -21287.882,E2 -21287.882} C_VEL
LIN {X 0,Y 248.519,Z 397.004,A -85,B 0,C 180,E1 -21288.566,E2 -21288.566} C_VEL
LIN {X 0,Y 243.847,Z 434.52,A -85,B 0,C 180,E1 -21290.013,E2 -21290.013} C_VEL
LIN {X 0,Y 241.131,Z 448.415,A -85,B 0,C 180,E1 -21290.803,E2 -21290.803} C_VEL
LIN {X 0,Y 237.42,Z 461.812,A -85,B 0,C 180,E1 -21291.843,E2 -21291.843} C_VEL
LIN {X 0,Y 233.104,Z 474.496,A -85,B 0,C 180,E1 -21293.194,E2 -21293.194} C_VEL
LIN {X 0,Y 227.999,Z 486.935,A -85,B 0,C 180,E1 -21294.97,E2 -21294.97} C_VEL
LIN {X 0,Y 223.826,Z 496.14,A -85,B 0,C 180,E1 -21296.675,E2 -21296.675} C_VEL
LIN {X 0,Y 219.488,Z 504.708,A -85,B 0,C 180,E1 -21298.653,E2 -21298.653} C_VEL
LIN {X 0,Y 214.67,Z 513.188,A -85,B 0,C 180,E1 -21301.132,E2 -21301.132} C_VEL
LIN {X 0,Y 209.904,Z 521.165,A -85,B 0,C 180,E1 -21304.204,E2 -21304.204} C_VEL
LIN {X 0,Y 206.187,Z 527.06,A -85,B 0,C 180,E1 -21307.177,E2 -21307.177} C_VEL
LIN {X 0,Y 203.559,Z 531.036,A -85,B 0,C 180,E1 -21309.808,E2 -21309.808} C_VEL
LIN {X 0,Y 201.935,Z 533.414,A -85,B 0,C 180,E1 -21311.751,E2 -21311.751} C_VEL
LIN {X 0,Y 199.256,Z 536.87,A -85,B 0,C 180,E1 -21315.711,E2 -21315.711} C_VEL
LIN {X 0,Y 197.919,Z 538.785,A -85,B 0,C 180,E1 -21319.777,E2 -21319.777} C_VEL
LIN {X 0,Y 197.576,Z 539.155,A -85,B 0,C 180,E1 -21321.824,E2 -21321.824} C_VEL
LIN {X 0,Y 197.476,Z 538.9,A -85,B 0,C 180,E1 -21325.212,E2 -21325.212} C_VEL
LIN {X 0,Y 197.627,Z 537.845,A -85,B 0,C 180,E1 -21327.965,E2 -21327.965} C_VEL
LIN {X 0,Y 197.811,Z 536.587,A -85,B 0,C 180,E1 -21330.003,E2 -21330.003} C_VEL
LIN {X 0,Y 197.763,Z 533.754,A -85,B 0,C 180,E1 -21333.059,E2 -21333.059} C_VEL
LIN {X 0,Y 197.848,Z 529.785,A -85,B 0,C 180,E1 -21336.12,E2 -21336.12} C_VEL
LIN {X 0,Y 198.086,Z 523.494,A -85,B 0,C 180,E1 -21339.705,E2 -21339.705} C_VEL
LIN {X 0,Y 198.718,Z 516.558,A -85,B 0,C 180,E1 -21342.772,E2 -21342.772} C_VEL
LIN {X 0,Y 199.679,Z 509.465,A -85,B 0,C 180,E1 -21345.308,E2 -21345.308} C_VEL
LIN {X 0,Y 200.868,Z 500.862,A -85,B 0,C 180,E1 -21347.829,E2 -21347.829} C_VEL
LIN {X 0,Y 202.528,Z 490.256,A -85,B 0,C 180,E1 -21350.306,E2 -21350.306} C_VEL
LIN {X 0,Y 204.092,Z 479.823,A -85,B 0,C 180,E1 -21352.26,E2 -21352.26} C_VEL
LIN {X 0,Y 205.661,Z 468.505,A -85,B 0,C 180,E1 -21353.942,E2 -21353.942} C_VEL
LIN {X 0,Y 207.34,Z 454.776,A -85,B 0,C 180,E1 -21355.472,E2 -21355.472} C_VEL
LIN {X 0,Y 208.622,Z 441.59,A -85,B 0,C 180,E1 -21356.511,E2 -21356.511} C_VEL
LIN {X 0,Y 209.546,Z 424.136,A -85,B 0,C 180,E1 -21357.395,E2 -21357.395} C_VEL
LIN {X 0,Y 211.279,Z 385.884,A -85,B 0,C 180,E1 -21359.101,E2 -21359.101} C_VEL
LIN {X 0,Y 207.244,Z 344.69,A -85,B 0,C 180,E1 -21361.475,E2 -21361.475} C_VEL
LIN {X 0,Y 202.381,Z 328.633,A -85,B 0,C 180,E1 -21362.8,E2 -21362.8} C_VEL
LIN {X 0,Y 200.302,Z 318.467,A -85,B 0,C 180,E1 -21367.247,E2 -21367.247} C_VEL
LIN {X 0,Y 199.684,Z 315.61,A -85,B 0,C 180,E1 -21368.624,E2 -21368.624} C_VEL
LIN {X 0,Y 199.564,Z 315.626,A -85,B 0,C 180,E1 -21372.305,E2 -21372.305} C_VEL
LIN {X 0,Y 199.574,Z 315.621,A -85,B 0,C 180,E1 -21375.226,E2 -21375.226} C_VEL
LIN {X 0,Y 199.567,Z 315.623,A -85,B 0,C 180,E1 -21378,E2 -21378} C_VEL
LIN {X 0,Y 199.594,Z 315.624,A -85,B 0,C 180,E1 -21380.771,E2 -21380.771} C_VEL
LIN {X 0,Y 199.604,Z 315.62,A -85,B 0,C 180,E1 -21385.711,E2 -21385.711} C_VEL
LIN {X 0,Y 199.677,Z 315.611,A -85,B 0,C 180,E1 -21388.132,E2 -21388.132} C_VEL
LIN {X 0,Y 199.635,Z 315.617,A -85,B 0,C 180,E1 -21392.763,E2 -21392.763} C_VEL
LIN {X 0,Y 199.67,Z 315.611,A -85,B 0,C 180,E1 -21397.22,E2 -21397.22} C_VEL
LIN {X 0,Y 199.739,Z 315.603,A -85,B 0,C 180,E1 -21401.801,E2 -21401.801} C_VEL
LIN {X 0,Y 199.789,Z 315.595,A -85,B 0,C 180,E1 -21405.744,E2 -21405.744} C_VEL
LIN {X 0,Y 200.015,Z 315.569,A -85,B 0,C 180,E1 -21409.88,E2 -21409.88} C_VEL
LIN {X 0,Y 200,Z 315.568,A -85,B 0,C 180,E1 -21413.948,E2 -21413.948} C_VEL
LIN {X 0,Y 200.301,Z 315.534,A -85,B 0,C 180,E1 -21417.988,E2 -21417.988} C_VEL
LIN {X 0,Y 200.455,Z 315.513,A -85,B 0,C 180,E1 -21419.999,E2 -21419.999} C_VEL
LIN {X 0,Y 199.998,Z 315.57,A -85,B 0,C 180,E1 -21424.029,E2 -21424.029} C_VEL
LIN {X 0,Y 200.063,Z 315.562,A -85,B 0,C 180,E1 -21428.077,E2 -21428.077} C_VEL
LIN {X 0,Y 199.849,Z 315.589,A -85,B 0,C 180,E1 -21432.18,E2 -21432.18} C_VEL
LIN {X 0,Y 199.738,Z 315.603,A -85,B 0,C 180,E1 -21436.348,E2 -21436.348} C_VEL
LIN {X 0,Y 199.634,Z 315.614,A -85,B 0,C 180,E1 -21440.611,E2 -21440.611} C_VEL
LIN {X 0,Y 199.652,Z 315.613,A -85,B 0,C 180,E1 -21444.986,E2 -21444.986} C_VEL
LIN {X 0,Y 199.656,Z 315.613,A -85,B 0,C 180,E1 -21449.524,E2 -21449.524} C_VEL
LIN {X 0,Y 199.663,Z 315.613,A -85,B 0,C 180,E1 -21452.355,E2 -21452.355} C_VEL
LIN {X 0,Y 199.616,Z 315.616,A -85,B 0,C 180,E1 -21456.763,E2 -21456.763} C_VEL
LIN {X 0,Y 199.601,Z 315.62,A -85,B 0,C 180,E1 -21459.328,E2 -21459.328} C_VEL
LIN {X 0,Y 199.57,Z 315.624,A -85,B 0,C 180,E1 -21462.31,E2 -21462.31} C_VEL
LIN {X 0,Y 199.61,Z 315.616,A -85,B 0,C 180,E1 -21465.238,E2 -21465.238} C_VEL
LIN {X 0,Y 199.65,Z 315.617,A -85,B 0,C 180,E1 -21468.024,E2 -21468.024} C_VEL
LIN {X 0,Y 199.676,Z 315.609,A -85,B 0,C 180,E1 -21470.743,E2 -21470.743} C_VEL
LIN {X 0,Y 199.63,Z 315.617,A -85,B 0,C 180,E1 -21475.717,E2 -21475.717} C_VEL
LIN {X 0,Y 199.693,Z 315.612,A -85,B 0,C 180,E1 -21478.136,E2 -21478.136} C_VEL
LIN {X 0,Y 199.684,Z 315.61,A -85,B 0,C 180,E1 -21482.771,E2 -21482.771} C_VEL
LIN {X 0,Y 199.737,Z 315.602,A -85,B 0,C 180,E1 -21487.228,E2 -21487.228} C_VEL
LIN {X 0,Y 199.795,Z 315.595,A -85,B 0,C 180,E1 -21491.756,E2 -21491.756} C_VEL
LIN {X 0,Y 199.835,Z 315.59,A -85,B 0,C 180,E1 -21495.746,E2 -21495.746} C_VEL
LIN {X 0,Y 200.074,Z 315.56,A -85,B 0,C 180,E1 -21499.882,E2 -21499.882} C_VEL
LIN {X 0,Y 200.131,Z 315.554,A -85,B 0,C 180,E1 -21501.923,E2 -21501.923} C_VEL
LIN {X 0,Y 200.32,Z 315.529,A -85,B 0,C 180,E1 -21507.986,E2 -21507.986} C_VEL
LIN {X 0,Y 200.477,Z 315.511,A -85,B 0,C 180,E1 -21509.997,E2 -21509.997} C_VEL
LIN {X 0,Y 200.029,Z 315.565,A -85,B 0,C 180,E1 -21514.026,E2 -21514.026} C_VEL
LIN {X 0,Y 200.12,Z 315.556,A -85,B 0,C 180,E1 -21518.071,E2 -21518.071} C_VEL
LIN {X 0,Y 199.909,Z 315.581,A -85,B 0,C 180,E1 -21522.173,E2 -21522.173} C_VEL
LIN {X 0,Y 199.807,Z 315.593,A -85,B 0,C 180,E1 -21526.338,E2 -21526.338} C_VEL
LIN {X 0,Y 199.739,Z 315.606,A -85,B 0,C 180,E1 -21530.595,E2 -21530.595} C_VEL
LIN {X 0,Y 199.666,Z 315.614,A -85,B 0,C 180,E1 -21534.979,E2 -21534.979} C_VEL
LIN {X 0,Y 199.682,Z 315.612,A -85,B 0,C 180,E1 -21539.552,E2 -21539.552} C_VEL
LIN {X 0,Y 212.464,Z 349.398,A -85,B 0,C 180,E1 -21542.487,E2 -21542.487} C_VEL
LIN {X 0,Y 209.07,Z 415.287,A -85,B 0,C 180,E1 -21545.426,E2 -21545.426} C_VEL
LIN {X 0,Y 208.129,Z 429.534,A -85,B 0,C 180,E1 -21546.481,E2 -21546.481} C_VEL
LIN {X 0,Y 206.802,Z 442.164,A -85,B 0,C 180,E1 -21547.807,E2 -21547.807} C_VEL
LIN {X 0,Y 205.512,Z 453.148,A -85,B 0,C 180,E1 -21549.313,E2 -21549.313} C_VEL
LIN {X 0,Y 203.777,Z 465.275,A -85,B 0,C 180,E1 -21551.413,E2 -21551.413} C_VEL
LIN {X 0,Y 202.245,Z 475.732,A -85,B 0,C 180,E1 -21553.718,E2 -21553.718} C_VEL
LIN {X 0,Y 200.9,Z 484.742,A -85,B 0,C 180,E1 -21556.158,E2 -21556.158} C_VEL
LIN {X 0,Y 199.728,Z 492.509,A -85,B 0,C 180,E1 -21558.719,E2 -21558.719} C_VEL
LIN {X 0,Y 198.62,Z 500.473,A -85,B 0,C 180,E1 -21561.989,E2 -21561.989} C_VEL
LIN {X 0,Y 197.904,Z 506.902,A -85,B 0,C 180,E1 -21565.377,E2 -21565.377} C_VEL
LIN {X 0,Y 197.435,Z 511.701,A -85,B 0,C 180,E1 -21568.669,E2 -21568.669} C_VEL
LIN {X 0,Y 197.275,Z 515.598,A -85,B 0,C 180,E1 -21572.412,E2 -21572.412} C_VEL
LIN {X 0,Y 197.486,Z 517.259,A -85,B 0,C 180,E1 -21574.721,E2 -21574.721} C_VEL
LIN {X 0,Y 197.979,Z 518.519,A -85,B 0,C 180,E1 -21577.341,E2 -21577.341} C_VEL
LIN {X 0,Y 198.528,Z 519.014,A -85,B 0,C 180,E1 -21579.269,E2 -21579.269} C_VEL
LIN {X 0,Y 199.594,Z 519.135,A -85,B 0,C 180,E1 -21581.908,E2 -21581.908} C_VEL
LIN {X 0,Y 201.867,Z 517.928,A -85,B 0,C 180,E1 -21585.896,E2 -21585.896} C_VEL
LIN {X 0,Y 203.426,Z 516.636,A -85,B 0,C 180,E1 -21588.037,E2 -21588.037} C_VEL
LIN {X 0,Y 206.233,Z 513.755,A -85,B 0,C 180,E1 -21591.155,E2 -21591.155} C_VEL
LIN {X 0,Y 209.656,Z 509.598,A -85,B 0,C 180,E1 -21594.229,E2 -21594.229} C_VEL
LIN {X 0,Y 214.297,Z 503.119,A -85,B 0,C 180,E1 -21597.651,E2 -21597.651} C_VEL
LIN {X 0,Y 218.895,Z 495.932,A -85,B 0,C 180,E1 -21600.461,E2 -21600.461} C_VEL
LIN {X 0,Y 223.094,Z 488.502,A -85,B 0,C 180,E1 -21602.709,E2 -21602.709} C_VEL
LIN {X 0,Y 227.836,Z 478.978,A -85,B 0,C 180,E1 -21604.971,E2 -21604.971} C_VEL
LIN {X 0,Y 232.436,Z 468.324,A -85,B 0,C 180,E1 -21606.948,E2 -21606.948} C_VEL
LIN {X 0,Y 236.471,Z 457.265,A -85,B 0,C 180,E1 -21608.547,E2 -21608.547} C_VEL
LIN {X 0,Y 240.127,Z 445.097,A -85,B 0,C 180,E1 -21609.902,E2 -21609.902} C_VEL
LIN {X 0,Y 243.114,Z 432.132,A -85,B 0,C 180,E1 -21610.98,E2 -21610.98} C_VEL
LIN {X 0,Y 245.35,Z 418.915,A -85,B 0,C 180,E1 -21611.753,E2 -21611.753} C_VEL
LIN {X 0,Y 250.105,Z 379.884,A -85,B 0,C 180,E1 -21613.292,E2 -21613.292} C_VEL
LIN {X 0,Y 247.693,Z 374.817,A -85,B 0,C 180,E1 -21614.865,E2 -21614.865} C_VEL
LIN {X 0,Y 244.519,Z 369.066,A -85,B 0,C 180,E1 -21617.21,E2 -21617.21} C_VEL
LIN {X 0,Y 241.926,Z 364.826,A -85,B 0,C 180,E1 -21619.482,E2 -21619.482} C_VEL
LIN {X 0,Y 238.97,Z 360.489,A -85,B 0,C 180,E1 -21622.842,E2 -21622.842} C_VEL
LIN {X 0,Y 236.523,Z 357.898,A -85,B 0,C 180,E1 -21627.396,E2 -21627.396} C_VEL
LIN {X 0,Y 236.016,Z 357.861,A -85,B 0,C 180,E1 -21631.029,E2 -21631.029} C_VEL
LIN {X 0,Y 236.615,Z 359.245,A -85,B 0,C 180,E1 -21634.358,E2 -21634.358} C_VEL
LIN {X 0,Y 238.491,Z 363.993,A -85,B 0,C 180,E1 -21638.358,E2 -21638.358} C_VEL
LIN {X 0,Y 239.715,Z 366.496,A -85,B 0,C 180,E1 -21640.035,E2 -21640.035} C_VEL
LIN {X 0,Y 242.26,Z 372.149,A -85,B 0,C 180,E1 -21642.777,E2 -21642.777} C_VEL
LIN {X 0,Y 244.446,Z 377.379,A -85,B 0,C 180,E1 -21644.691,E2 -21644.691} C_VEL
LIN {X 0,Y 246.718,Z 383.363,A -85,B 0,C 180,E1 -21646.495,E2 -21646.495} C_VEL
LIN {X 0,Y 247.302,Z 385.105,A -85,B 0,C 180,E1 -21646.932,E2 -21646.932} C_VEL
LIN {X 0,Y 247.628,Z 387.717,A -85,B 0,C 180,E1 -21647.326,E2 -21647.326} C_VEL
LIN {X 0,Y 247.291,Z 391.488,A -85,B 0,C 180,E1 -21647.529,E2 -21647.529} C_VEL
LIN {X 0,Y 245.932,Z 397.559,A -85,B 0,C 180,E1 -21647.492,E2 -21647.492} C_VEL
LIN {X 0,Y 244.269,Z 404.616,A -85,B 0,C 180,E1 -21647.411,E2 -21647.411} C_VEL
LIN {X 0,Y 244.04,Z 406.039,A -85,B 0,C 180,E1 -21647.442,E2 -21647.442} C_VEL
LIN {X 0,Y 240.232,Z 434.507,A -85,B 0,C 180,E1 -21648.564,E2 -21648.564} C_VEL
LIN {X 0,Y 237.342,Z 448.302,A -85,B 0,C 180,E1 -21649.358,E2 -21649.358} C_VEL
LIN {X 0,Y 233.807,Z 460.584,A -85,B 0,C 180,E1 -21650.31,E2 -21650.31} C_VEL
LIN {X 0,Y 229.798,Z 472.017,A -85,B 0,C 180,E1 -21651.463,E2 -21651.463} C_VEL
LIN {X 0,Y 224.987,Z 483.749,A -85,B 0,C 180,E1 -21653.044,E2 -21653.044} C_VEL
LIN {X 0,Y 220.898,Z 492.375,A -85,B 0,C 180,E1 -21654.513,E2 -21654.513} C_VEL
LIN {X 0,Y 215.307,Z 502.974,A -85,B 0,C 180,E1 -21656.863,E2 -21656.863} C_VEL
LIN {X 0,Y 210.169,Z 511.727,A -85,B 0,C 180,E1 -21659.346,E2 -21659.346} C_VEL
LIN {X 0,Y 205.663,Z 518.834,A -85,B 0,C 180,E1 -21661.981,E2 -21661.981} C_VEL
LIN {X 0,Y 201.087,Z 525.472,A -85,B 0,C 180,E1 -21665.209,E2 -21665.209} C_VEL
LIN {X 0,Y 197.832,Z 529.992,A -85,B 0,C 180,E1 -21668.104,E2 -21668.104} C_VEL
LIN {X 0,Y 195.193,Z 533.511,A -85,B 0,C 180,E1 -21671.098,E2 -21671.098} C_VEL
LIN {X 0,Y 192.351,Z 536.754,A -85,B 0,C 180,E1 -21675.186,E2 -21675.186} C_VEL
LIN {X 0,Y 191.509,Z 537.802,A -85,B 0,C 180,E1 -21677.285,E2 -21677.285} C_VEL
LIN {X 0,Y 190.538,Z 538.693,A -85,B 0,C 180,E1 -21681.52,E2 -21681.52} C_VEL
LIN {X 0,Y 190.431,Z 538.23,A -85,B 0,C 180,E1 -21685.186,E2 -21685.186} C_VEL
LIN {X 0,Y 190.559,Z 537.137,A -85,B 0,C 180,E1 -21687.89,E2 -21687.89} C_VEL
LIN {X 0,Y 190.75,Z 535.753,A -85,B 0,C 180,E1 -21690.003,E2 -21690.003} C_VEL
LIN {X 0,Y 190.718,Z 532.761,A -85,B 0,C 180,E1 -21693.172,E2 -21693.172} C_VEL
LIN {X 0,Y 190.798,Z 528.6,A -85,B 0,C 180,E1 -21696.347,E2 -21696.347} C_VEL
LIN {X 0,Y 191.093,Z 522.101,A -85,B 0,C 180,E1 -21700.063,E2 -21700.063} C_VEL
LIN {X 0,Y 191.782,Z 514.897,A -85,B 0,C 180,E1 -21703.242,E2 -21703.242} C_VEL
LIN {X 0,Y 193.085,Z 505.883,A -85,B 0,C 180,E1 -21706.387,E2 -21706.387} C_VEL
LIN {X 0,Y 194.405,Z 496.584,A -85,B 0,C 180,E1 -21708.989,E2 -21708.989} C_VEL
LIN {X 0,Y 196.228,Z 485.315,A -85,B 0,C 180,E1 -21711.483,E2 -21711.483} C_VEL
LIN {X 0,Y 197.974,Z 473.53,A -85,B 0,C 180,E1 -21713.54,E2 -21713.54} C_VEL
LIN {X 0,Y 199.713,Z 460.511,A -85,B 0,C 180,E1 -21715.258,E2 -21715.258} C_VEL
LIN {X 0,Y 201.071,Z 448.244,A -85,B 0,C 180,E1 -21716.466,E2 -21716.466} C_VEL
LIN {X 0,Y 202.027,Z 436.102,A -85,B 0,C 180,E1 -21717.308,E2 -21717.308} C_VEL
LIN {X 0,Y 204.498,Z 386.668,A -85,B 0,C 180,E1 -21719.624,E2 -21719.624} C_VEL
LIN {X 0,Y 200.62,Z 346.413,A -85,B 0,C 180,E1 -21722.013,E2 -21722.013} C_VEL
LIN {X 0,Y 195.081,Z 328.251,A -85,B 0,C 180,E1 -21723.573,E2 -21723.573} C_VEL
LIN {X 0,Y 192.752,Z 317.057,A -85,B 0,C 180,E1 -21728.701,E2 -21728.701} C_VEL
LIN {X 0,Y 192.623,Z 316.49,A -85,B 0,C 180,E1 -21728.971,E2 -21728.971} C_VEL
LIN {X 0,Y 192.485,Z 316.507,A -85,B 0,C 180,E1 -21733.925,E2 -21733.925} C_VEL
LIN {X 0,Y 192.502,Z 316.507,A -85,B 0,C 180,E1 -21738.915,E2 -21738.915} C_VEL
LIN {X 0,Y 192.579,Z 316.496,A -85,B 0,C 180,E1 -21743.403,E2 -21743.403} C_VEL
LIN {X 0,Y 192.6,Z 316.495,A -85,B 0,C 180,E1 -21747.061,E2 -21747.061} C_VEL
LIN {X 0,Y 192.612,Z 316.491,A -85,B 0,C 180,E1 -21751.682,E2 -21751.682} C_VEL
LIN {X 0,Y 192.663,Z 316.482,A -85,B 0,C 180,E1 -21756.342,E2 -21756.342} C_VEL
LIN {X 0,Y 192.688,Z 316.483,A -85,B 0,C 180,E1 -21761.491,E2 -21761.491} C_VEL
LIN {X 0,Y 192.716,Z 316.477,A -85,B 0,C 180,E1 -21765.209,E2 -21765.209} C_VEL
LIN {X 0,Y 192.939,Z 316.452,A -85,B 0,C 180,E1 -21769.566,E2 -21769.566} C_VEL
LIN {X 0,Y 192.963,Z 316.445,A -85,B 0,C 180,E1 -21773.726,E2 -21773.726} C_VEL
LIN {X 0,Y 193.243,Z 316.413,A -85,B 0,C 180,E1 -21777.915,E2 -21777.915} C_VEL
LIN {X 0,Y 193.42,Z 316.389,A -85,B 0,C 180,E1 -21779.999,E2 -21779.999} C_VEL
LIN {X 0,Y 192.944,Z 316.449,A -85,B 0,C 180,E1 -21784.177,E2 -21784.177} C_VEL
LIN {X 0,Y 193.014,Z 316.44,A -85,B 0,C 180,E1 -21788.374,E2 -21788.374} C_VEL
LIN {X 0,Y 192.775,Z 316.469,A -85,B 0,C 180,E1 -21792.634,E2 -21792.634} C_VEL
LIN {X 0,Y 192.697,Z 316.479,A -85,B 0,C 180,E1 -21796.963,E2 -21796.963} C_VEL
LIN {X 0,Y 192.571,Z 316.496,A -85,B 0,C 180,E1 -21801.404,E2 -21801.404} C_VEL
LIN {X 0,Y 192.631,Z 316.489,A -85,B 0,C 180,E1 -21804.206,E2 -21804.206} C_VEL
LIN {X 0,Y 192.636,Z 316.486,A -85,B 0,C 180,E1 -21808.888,E2 -21808.888} C_VEL
LIN {X 0,Y 192.59,Z 316.493,A -85,B 0,C 180,E1 -21813.186,E2 -21813.186} C_VEL
LIN {X 0,Y 192.545,Z 316.5,A -85,B 0,C 180,E1 -21818.352,E2 -21818.352} C_VEL
LIN {X 0,Y 192.513,Z 316.501,A -85,B 0,C 180,E1 -21823.104,E2 -21823.104} C_VEL
LIN {X 0,Y 192.559,Z 316.497,A -85,B 0,C 180,E1 -21826.881,E2 -21826.881} C_VEL
LIN {X 0,Y 192.597,Z 316.492,A -85,B 0,C 180,E1 -21831.659,E2 -21831.659} C_VEL
LIN {X 0,Y 192.596,Z 316.493,A -85,B 0,C 180,E1 -21836.813,E2 -21836.813} C_VEL
LIN {X 0,Y 192.659,Z 316.481,A -85,B 0,C 180,E1 -21841.69,E2 -21841.69} C_VEL
LIN {X 0,Y 192.705,Z 316.482,A -85,B 0,C 180,E1 -21846.347,E2 -21846.347} C_VEL
LIN {X 0,Y 192.731,Z 316.474,A -85,B 0,C 180,E1 -21851.456,E2 -21851.456} C_VEL
LIN {X 0,Y 192.763,Z 316.471,A -85,B 0,C 180,E1 -21855.212,E2 -21855.212} C_VEL
LIN {X 0,Y 193.019,Z 316.438,A -85,B 0,C 180,E1 -21859.508,E2 -21859.508} C_VEL
LIN {X 0,Y 193.003,Z 316.442,A -85,B 0,C 180,E1 -21863.726,E2 -21863.726} C_VEL
LIN {X 0,Y 193.262,Z 316.408,A -85,B 0,C 180,E1 -21867.913,E2 -21867.913} C_VEL
LIN {X 0,Y 193.441,Z 316.388,A -85,B 0,C 180,E1 -21869.997,E2 -21869.997} C_VEL
LIN {X 0,Y 192.976,Z 316.444,A -85,B 0,C 180,E1 -21874.173,E2 -21874.173} C_VEL
LIN {X 0,Y 193.068,Z 316.436,A -85,B 0,C 180,E1 -21878.368,E2 -21878.368} C_VEL
LIN {X 0,Y 192.849,Z 316.463,A -85,B 0,C 180,E1 -21882.626,E2 -21882.626} C_VEL
LIN {X 0,Y 192.774,Z 316.471,A -85,B 0,C 180,E1 -21888.582,E2 -21888.582} C_VEL
LIN {X 0,Y 192.659,Z 316.486,A -85,B 0,C 180,E1 -21894.224,E2 -21894.224} C_VEL
LIN {X 0,Y 192.654,Z 316.487,A -85,B 0,C 180,E1 -21898.813,E2 -21898.813} C_VEL
LIN {X 0,Y 195.058,Z 323.107,A -85,B 0,C 180,E1 -21899.476,E2 -21899.476} C_VEL
LIN {X 0,Y 205.773,Z 351.35,A -85,B 0,C 180,E1 -21901.984,E2 -21901.984} C_VEL
LIN {X 0,Y 202.179,Z 415.567,A -85,B 0,C 180,E1 -21904.956,E2 -21904.956} C_VEL
LIN {X 0,Y 201.322,Z 428.783,A -85,B 0,C 180,E1 -21905.959,E2 -21905.959} C_VEL
LIN {X 0,Y 199.934,Z 441.692,A -85,B 0,C 180,E1 -21907.318,E2 -21907.318} C_VEL
LIN {X 0,Y 198.344,Z 454.395,A -85,B 0,C 180,E1 -21909.116,E2 -21909.116} C_VEL
LIN {X 0,Y 196.808,Z 465.188,A -85,B 0,C 180,E1 -21911.058,E2 -21911.058} C_VEL
LIN {X 0,Y 195.21,Z 475.9,A -85,B 0,C 180,E1 -21913.481,E2 -21913.481} C_VEL
LIN {X 0,Y 193.636,Z 486.246,A -85,B 0,C 180,E1 -21916.403,E2 -21916.403} C_VEL
LIN {X 0,Y 192.261,Z 495.273,A -85,B 0,C 180,E1 -21919.642,E2 -21919.642} C_VEL
LIN {X 0,Y 191.357,Z 502.092,A -85,B 0,C 180,E1 -21922.701,E2 -21922.701} C_VEL
LIN {X 0,Y 190.832,Z 506.674,A -85,B 0,C 180,E1 -21925.228,E2 -21925.228} C_VEL
LIN {X 0,Y 190.308,Z 511.881,A -85,B 0,C 180,E1 -21928.869,E2 -21928.869} C_VEL
LIN {X 0,Y 190.179,Z 515.638,A -85,B 0,C 180,E1 -21932.469,E2 -21932.469} C_VEL
LIN {X 0,Y 190.823,Z 518.554,A -85,B 0,C 180,E1 -21937.013,E2 -21937.013} C_VEL
LIN {X 0,Y 191.959,Z 519.582,A -85,B 0,C 180,E1 -21940.762,E2 -21940.762} C_VEL
LIN {X 0,Y 193.026,Z 519.56,A -85,B 0,C 180,E1 -21943.067,E2 -21943.067} C_VEL
LIN {X 0,Y 195.11,Z 518.617,A -85,B 0,C 180,E1 -21946.508,E2 -21946.508} C_VEL
LIN {X 0,Y 197.664,Z 516.642,A -85,B 0,C 180,E1 -21949.761,E2 -21949.761} C_VEL
LIN {X 0,Y 200.831,Z 513.513,A -85,B 0,C 180,E1 -21952.966,E2 -21952.966} C_VEL
LIN {X 0,Y 204.698,Z 509.168,A -85,B 0,C 180,E1 -21956.064,E2 -21956.064} C_VEL
LIN {X 0,Y 208.982,Z 503.546,A -85,B 0,C 180,E1 -21959.037,E2 -21959.037} C_VEL
LIN {X 0,Y 213.883,Z 496.307,A -85,B 0,C 180,E1 -21961.884,E2 -21961.884} C_VEL
LIN {X 0,Y 219.088,Z 487.601,A -85,B 0,C 180,E1 -21964.489,E2 -21964.489} C_VEL
LIN {X 0,Y 224.159,Z 477.831,A -85,B 0,C 180,E1 -21966.753,E2 -21966.753} C_VEL
LIN {X 0,Y 228.631,Z 467.744,A -85,B 0,C 180,E1 -21968.566,E2 -21968.566} C_VEL
LIN {X 0,Y 233.049,Z 455.988,A -85,B 0,C 180,E1 -21970.206,E2 -21970.206} C_VEL
LIN {X 0,Y 236.87,Z 443.493,A -85,B 0,C 180,E1 -21971.535,E2 -21971.535} C_VEL
LIN {X 0,Y 239.892,Z 430.714,A -85,B 0,C 180,E1 -21972.56,E2 -21972.56} C_VEL
LIN {X 0,Y 242.202,Z 416.802,A -85,B 0,C 180,E1 -21973.32,E2 -21973.32} C_VEL
LIN {X 0,Y 246.383,Z 383.481,A -85,B 0,C 180,E1 -21974.631,E2 -21974.631} C_VEL
LIN {X 0,Y 244.261,Z 378.978,A -85,B 0,C 180,E1 -21976.209,E2 -21976.209} C_VEL
LIN {X 0,Y 241.366,Z 373.725,A -85,B 0,C 180,E1 -21978.602,E2 -21978.602} C_VEL
LIN {X 0,Y 239.322,Z 370.374,A -85,B 0,C 180,E1 -21980.635,E2 -21980.635} C_VEL
LIN {X 0,Y 237.224,Z 367.175,A -85,B 0,C 180,E1 -21983.326,E2 -21983.326} C_VEL
LIN {X 0,Y 235.145,Z 364.833,A -85,B 0,C 180,E1 -21987.57,E2 -21987.57} C_VEL
LIN {X 0,Y 234.662,Z 364.756,A -85,B 0,C 180,E1 -21990.607,E2 -21990.607} C_VEL
LIN {X 0,Y 235.151,Z 366.078,A -85,B 0,C 180,E1 -21994.034,E2 -21994.034} C_VEL
LIN {X 0,Y 236.748,Z 370.514,A -85,B 0,C 180,E1 -21997.843,E2 -21997.843} C_VEL
LIN {X 0,Y 237.847,Z 373.026,A -85,B 0,C 180,E1 -21999.505,E2 -21999.505} C_VEL
LIN {X 0,Y 240.15,Z 378.501,A -85,B 0,C 180,E1 -22002.189,E2 -22002.189} C_VEL
LIN {X 0,Y 242.032,Z 383.465,A -85,B 0,C 180,E1 -22004.023,E2 -22004.023} C_VEL
LIN {X 0,Y 244,Z 389.179,A -85,B 0,C 180,E1 -22005.761,E2 -22005.761} C_VEL
LIN {X 0,Y 245.097,Z 392.74,A -85,B 0,C 180,E1 -22006.652,E2 -22006.652} C_VEL
LIN {X 0,Y 245.042,Z 397.96,A -85,B 0,C 180,E1 -22007.129,E2 -22007.129} C_VEL
LIN {X 0,Y 244.04,Z 406.039,A -85,B 0,C 180,E1 -22007.442,E2 -22007.442} C_VEL
LIN {X 0,Y 242.961,Z 411.857,A -85,B 0,C 180,E1 -22007.496,E2 -22007.496} C_VEL
LIN {X 0,Y 237.771,Z 430.909,A -85,B 0,C 180,E1 -22007.023,E2 -22007.023} C_VEL
LIN {X 0,Y 236.461,Z 436.627,A -85,B 0,C 180,E1 -22007.156,E2 -22007.156} C_VEL
LIN {X 0,Y 233.121,Z 450.831,A -85,B 0,C 180,E1 -22008.027,E2 -22008.027} C_VEL
LIN {X 0,Y 229.139,Z 463.389,A -85,B 0,C 180,E1 -22009.044,E2 -22009.044} C_VEL
LIN {X 0,Y 224.465,Z 475.37,A -85,B 0,C 180,E1 -22010.37,E2 -22010.37} C_VEL
LIN {X 0,Y 218.942,Z 487.386,A -85,B 0,C 180,E1 -22012.136,E2 -22012.136} C_VEL
LIN {X 0,Y 213.357,Z 498.041,A -85,B 0,C 180,E1 -22014.227,E2 -22014.227} C_VEL
LIN {X 0,Y 207.699,Z 507.552,A -85,B 0,C 180,E1 -22016.65,E2 -22016.65} C_VEL
LIN {X 0,Y 202.492,Z 515.28,A -85,B 0,C 180,E1 -22019.214,E2 -22019.214} C_VEL
LIN {X 0,Y 197.299,Z 522.573,A -85,B 0,C 180,E1 -22022.421,E2 -22022.421} C_VEL
LIN {X 0,Y 193.859,Z 527.087,A -85,B 0,C 180,E1 -22025.005,E2 -22025.005} C_VEL
LIN {X 0,Y 190.262,Z 531.498,A -85,B 0,C 180,E1 -22028.328,E2 -22028.328} C_VEL
LIN {X 0,Y 186.817,Z 535.324,A -85,B 0,C 180,E1 -22032.49,E2 -22032.49} C_VEL
LIN {X 0,Y 185.469,Z 536.619,A -85,B 0,C 180,E1 -22034.623,E2 -22034.623} C_VEL
LIN {X 0,Y 183.903,Z 538.064,A -85,B 0,C 180,E1 -22038.989,E2 -22038.989} C_VEL
LIN {X 0,Y 183.357,Z 538.024,A -85,B 0,C 180,E1 -22043.401,E2 -22043.401} C_VEL
LIN {X 0,Y 183.398,Z 537.393,A -85,B 0,C 180,E1 -22045.608,E2 -22045.608} C_VEL
LIN {X 0,Y 183.499,Z 536.338,A -85,B 0,C 180,E1 -22047.809,E2 -22047.809} C_VEL
LIN {X 0,Y 183.711,Z 534.867,A -85,B 0,C 180,E1 -22050.004,E2 -22050.004} C_VEL
LIN {X 0,Y 183.697,Z 531.718,A -85,B 0,C 180,E1 -22053.293,E2 -22053.293} C_VEL
LIN {X 0,Y 183.737,Z 528.265,A -85,B 0,C 180,E1 -22055.998,E2 -22055.998} C_VEL
LIN {X 0,Y 183.941,Z 522.767,A -85,B 0,C 180,E1 -22059.348,E2 -22059.348} C_VEL
LIN {X 0,Y 184.535,Z 515.849,A -85,B 0,C 180,E1 -22062.652,E2 -22062.652} C_VEL
LIN {X 0,Y 185.486,Z 508.771,A -85,B 0,C 180,E1 -22065.382,E2 -22065.382} C_VEL
LIN {X 0,Y 186.734,Z 500.203,A -85,B 0,C 180,E1 -22068.091,E2 -22068.091} C_VEL
LIN {X 0,Y 188.561,Z 489.032,A -85,B 0,C 180,E1 -22070.892,E2 -22070.892} C_VEL
LIN {X 0,Y 190.282,Z 477.878,A -85,B 0,C 180,E1 -22073.107,E2 -22073.107} C_VEL
LIN {X 0,Y 191.92,Z 466.212,A -85,B 0,C 180,E1 -22074.906,E2 -22074.906} C_VEL
LIN {X 0,Y 193.587,Z 453.406,A -85,B 0,C 180,E1 -22076.407,E2 -22076.407} C_VEL
LIN {X 0,Y 194.922,Z 440.01,A -85,B 0,C 180,E1 -22077.514,E2 -22077.514} C_VEL
LIN {X 0,Y 195.882,Z 422.434,A -85,B 0,C 180,E1 -22078.459,E2 -22078.459} C_VEL
LIN {X 0,Y 197.725,Z 387.794,A -85,B 0,C 180,E1 -22080.118,E2 -22080.118} C_VEL
LIN {X 0,Y 193.881,Z 347.733,A -85,B 0,C 180,E1 -22082.599,E2 -22082.599} C_VEL
LIN {X 0,Y 187.748,Z 327.838,A -85,B 0,C 180,E1 -22084.411,E2 -22084.411} C_VEL
LIN {X 0,Y 185.568,Z 317.474,A -85,B 0,C 180,E1 -22089.35,E2 -22089.35} C_VEL
LIN {X 0,Y 185.454,Z 317.383,A -85,B 0,C 180,E1 -22093.942,E2 -22093.942} C_VEL
LIN {X 0,Y 185.459,Z 317.384,A -85,B 0,C 180,E1 -22099.278,E2 -22099.278} C_VEL
LIN {X 0,Y 185.499,Z 317.377,A -85,B 0,C 180,E1 -22102.713,E2 -22102.713} C_VEL
LIN {X 0,Y 185.525,Z 317.374,A -85,B 0,C 180,E1 -22107.97,E2 -22107.97} C_VEL
LIN {X 0,Y 185.5,Z 317.379,A -85,B 0,C 180,E1 -22112.957,E2 -22112.957} C_VEL
LIN {X 0,Y 185.577,Z 317.366,A -85,B 0,C 180,E1 -22115.38,E2 -22115.38} C_VEL
LIN {X 0,Y 185.619,Z 317.365,A -85,B 0,C 180,E1 -22121.178,E2 -22121.178} C_VEL
LIN {X 0,Y 185.7,Z 317.35,A -85,B 0,C 180,E1 -22126.874,E2 -22126.874} C_VEL
LIN {X 0,Y 185.966,Z 317.321,A -85,B 0,C 180,E1 -22131.304,E2 -22131.304} C_VEL
LIN {X 0,Y 186.187,Z 317.292,A -85,B 0,C 180,E1 -22137.836,E2 -22137.836} C_VEL
LIN {X 0,Y 186.385,Z 317.266,A -85,B 0,C 180,E1 -22139.999,E2 -22139.999} C_VEL
LIN {X 0,Y 185.892,Z 317.327,A -85,B 0,C 180,E1 -22144.335,E2 -22144.335} C_VEL
LIN {X 0,Y 185.964,Z 317.318,A -85,B 0,C 180,E1 -22148.694,E2 -22148.694} C_VEL
LIN {X 0,Y 185.7,Z 317.351,A -85,B 0,C 180,E1 -22153.124,E2 -22153.124} C_VEL
LIN {X 0,Y 185.617,Z 317.358,A -85,B 0,C 180,E1 -22158.82,E2 -22158.82} C_VEL
LIN {X 0,Y 185.571,Z 317.367,A -85,B 0,C 180,E1 -22164.646,E2 -22164.646} C_VEL
LIN {X 0,Y 185.571,Z 317.367,A -85,B 0,C 180,E1 -22169.493,E2 -22169.493} C_VEL
LIN {X 0,Y 185.492,Z 317.375,A -85,B 0,C 180,E1 -22174.632,E2 -22174.632} C_VEL
LIN {X 0,Y 185.499,Z 317.374,A -85,B 0,C 180,E1 -22177.313,E2 -22177.313} C_VEL
LIN {X 0,Y 185.466,Z 317.381,A -85,B 0,C 180,E1 -22180.724,E2 -22180.724} C_VEL
LIN {X 0,Y 185.513,Z 317.375,A -85,B 0,C 180,E1 -22186.036,E2 -22186.036} C_VEL
LIN {X 0,Y 185.535,Z 317.375,A -85,B 0,C 180,E1 -22189.913,E2 -22189.913} C_VEL
LIN {X 0,Y 185.557,Z 317.366,A -85,B 0,C 180,E1 -22192.699,E2 -22192.699} C_VEL
LIN {X 0,Y 185.538,Z 317.374,A -85,B 0,C 180,E1 -22197.973,E2 -22197.973} C_VEL
LIN {X 0,Y 185.579,Z 317.364,A -85,B 0,C 180,E1 -22200.576,E2 -22200.576} C_VEL
LIN {X 0,Y 185.586,Z 317.366,A -85,B 0,C 180,E1 -22205.381,E2 -22205.381} C_VEL
LIN {X 0,Y 185.606,Z 317.36,A -85,B 0,C 180,E1 -22210.074,E2 -22210.074} C_VEL
LIN {X 0,Y 185.694,Z 317.354,A -85,B 0,C 180,E1 -22214.635,E2 -22214.635} C_VEL
LIN {X 0,Y 185.939,Z 317.32,A -85,B 0,C 180,E1 -22219.33,E2 -22219.33} C_VEL
LIN {X 0,Y 185.967,Z 317.318,A -85,B 0,C 180,E1 -22223.487,E2 -22223.487} C_VEL
LIN {X 0,Y 186.206,Z 317.286,A -85,B 0,C 180,E1 -22227.834,E2 -22227.834} C_VEL
LIN {X 0,Y 186.405,Z 317.264,A -85,B 0,C 180,E1 -22229.997,E2 -22229.997} C_VEL
LIN {X 0,Y 185.924,Z 317.323,A -85,B 0,C 180,E1 -22234.332,E2 -22234.332} C_VEL
LIN {X 0,Y 186.019,Z 317.316,A -85,B 0,C 180,E1 -22238.688,E2 -22238.688} C_VEL
LIN {X 0,Y 185.761,Z 317.346,A -85,B 0,C 180,E1 -22243.116,E2 -22243.116} C_VEL
LIN {X 0,Y 185.713,Z 317.349,A -85,B 0,C 180,E1 -22247.617,E2 -22247.617} C_VEL
LIN {X 0,Y 185.61,Z 317.363,A -85,B 0,C 180,E1 -22252.244,E2 -22252.244} C_VEL
LIN {X 0,Y 185.55,Z 317.374,A -85,B 0,C 180,E1 -22257.027,E2 -22257.027} C_VEL
LIN {X 0,Y 185.595,Z 317.365,A -85,B 0,C 180,E1 -22258.091,E2 -22258.091} C_VEL
LIN {X 0,Y 191.183,Z 332.023,A -85,B 0,C 180,E1 -22259.535,E2 -22259.535} C_VEL
LIN {X 0,Y 198.875,Z 352.496,A -85,B 0,C 180,E1 -22261.409,E2 -22261.409} C_VEL
LIN {X 0,Y 195.28,Z 416.158,A -85,B 0,C 180,E1 -22264.478,E2 -22264.478} C_VEL
LIN {X 0,Y 194.321,Z 429.711,A -85,B 0,C 180,E1 -22265.549,E2 -22265.549} C_VEL
LIN {X 0,Y 193.078,Z 441.215,A -85,B 0,C 180,E1 -22266.796,E2 -22266.796} C_VEL
LIN {X 0,Y 191.511,Z 453.696,A -85,B 0,C 180,E1 -22268.59,E2 -22268.59} C_VEL
LIN {X 0,Y 189.856,Z 464.893,A -85,B 0,C 180,E1 -22270.638,E2 -22270.638} C_VEL
LIN {X 0,Y 188.335,Z 474.973,A -85,B 0,C 180,E1 -22272.937,E2 -22272.937} C_VEL
LIN {X 0,Y 186.852,Z 484.377,A -85,B 0,C 180,E1 -22275.603,E2 -22275.603} C_VEL
LIN {X 0,Y 185.395,Z 493.803,A -85,B 0,C 180,E1 -22278.925,E2 -22278.925} C_VEL
LIN {X 0,Y 184.31,Z 501.549,A -85,B 0,C 180,E1 -22282.405,E2 -22282.405} C_VEL
LIN {X 0,Y 183.562,Z 508.273,A -85,B 0,C 180,E1 -22286.281,E2 -22286.281} C_VEL
LIN {X 0,Y 183.129,Z 513.191,A -85,B 0,C 180,E1 -22290.074,E2 -22290.074} C_VEL
LIN {X 0,Y 183.087,Z 515.651,A -85,B 0,C 180,E1 -22292.573,E2 -22292.573} C_VEL
LIN {X 0,Y 183.633,Z 518.518,A -85,B 0,C 180,E1 -22296.689,E2 -22296.689} C_VEL
LIN {X 0,Y 184.539,Z 519.748,A -85,B 0,C 180,E1 -22299.956,E2 -22299.956} C_VEL
LIN {X 0,Y 185.505,Z 520.084,A -85,B 0,C 180,E1 -22302.358,E2 -22302.358} C_VEL
LIN {X 0,Y 187.903,Z 519.516,A -85,B 0,C 180,E1 -22306.484,E2 -22306.484} C_VEL
LIN {X 0,Y 190.059,Z 518.221,A -85,B 0,C 180,E1 -22309.346,E2 -22309.346} C_VEL
LIN {X 0,Y 193.226,Z 515.682,A -85,B 0,C 180,E1 -22312.687,E2 -22312.687} C_VEL
LIN {X 0,Y 197.223,Z 511.782,A -85,B 0,C 180,E1 -22316.043,E2 -22316.043} C_VEL
LIN {X 0,Y 201.353,Z 507.009,A -85,B 0,C 180,E1 -22319.001,E2 -22319.001} C_VEL
LIN {X 0,Y 206.343,Z 500.623,A -85,B 0,C 180,E1 -22321.953,E2 -22321.953} C_VEL
LIN {X 0,Y 211.483,Z 493.092,A -85,B 0,C 180,E1 -22324.58,E2 -22324.58} C_VEL
LIN {X 0,Y 216.823,Z 484.136,A -85,B 0,C 180,E1 -22326.983,E2 -22326.983} C_VEL
LIN {X 0,Y 222.07,Z 473.917,A -85,B 0,C 180,E1 -22329.106,E2 -22329.106} C_VEL
LIN {X 0,Y 226.455,Z 463.961,A -85,B 0,C 180,E1 -22330.733,E2 -22330.733} C_VEL
LIN {X 0,Y 230.413,Z 453.382,A -85,B 0,C 180,E1 -22332.087,E2 -22332.087} C_VEL
LIN {X 0,Y 234.224,Z 440.72,A -85,B 0,C 180,E1 -22333.337,E2 -22333.337} C_VEL
LIN {X 0,Y 237.37,Z 426.744,A -85,B 0,C 180,E1 -22334.332,E2 -22334.332} C_VEL
LIN {X 0,Y 239.572,Z 412.571,A -85,B 0,C 180,E1 -22335.001,E2 -22335.001} C_VEL
LIN {X 0,Y 242.952,Z 387.33,A -85,B 0,C 180,E1 -22335.99,E2 -22335.99} C_VEL
LIN {X 0,Y 239.824,Z 381.103,A -85,B 0,C 180,E1 -22338.647,E2 -22338.647} C_VEL
LIN {X 0,Y 237.684,Z 377.232,A -85,B 0,C 180,E1 -22340.857,E2 -22340.857} C_VEL
LIN {X 0,Y 235.632,Z 374.001,A -85,B 0,C 180,E1 -22343.619,E2 -22343.619} C_VEL
LIN {X 0,Y 233.756,Z 371.775,A -85,B 0,C 180,E1 -22347.748,E2 -22347.748} C_VEL
LIN {X 0,Y 233.344,Z 371.859,A -85,B 0,C 180,E1 -22351.132,E2 -22351.132} C_VEL
LIN {X 0,Y 233.695,Z 373.017,A -85,B 0,C 180,E1 -22353.784,E2 -22353.784} C_VEL
LIN {X 0,Y 235.263,Z 377.61,A -85,B 0,C 180,E1 -22357.733,E2 -22357.733} C_VEL
LIN {X 0,Y 236.094,Z 379.75,A -85,B 0,C 180,E1 -22359.075,E2 -22359.075} C_VEL
LIN {X 0,Y 237.969,Z 384.561,A -85,B 0,C 180,E1 -22361.477,E2 -22361.477} C_VEL
LIN {X 0,Y 239.611,Z 389.443,A -85,B 0,C 180,E1 -22363.309,E2 -22363.309} C_VEL
LIN {X 0,Y 241.496,Z 395.46,A -85,B 0,C 180,E1 -22365.106,E2 -22365.106} C_VEL
LIN {X 0,Y 241.826,Z 397.022,A -85,B 0,C 180,E1 -22365.461,E2 -22365.461} C_VEL
LIN {X 0,Y 241.579,Z 400.617,A -85,B 0,C 180,E1 -22365.726,E2 -22365.726} C_VEL
